C05479=1163.449,223.532,-63.405,-177.710,7.285,148.703
C05480=1163.454,223.284,-63.379,-177.713,7.282,148.703
C05481=1163.458,223.036,-63.354,-177.715,7.280,148.703
C05482=1163.463,222.787,-63.329,-177.718,7.278,148.704
C05483=1163.468,222.538,-63.303,-177.721,7.275,148.704
C05484=1163.472,222.289,-63.277,-177.724,7.273,148.704
C05485=1163.477,222.041,-63.252,-177.726,7.271,148.704
C05486=1163.481,221.792,-63.227,-177.729,7.268,148.704
C05487=1163.486,221.544,-63.202,-177.732,7.265,148.705
C05488=1163.489,221.295,-63.177,-177.734,7.263,148.705
C05489=1163.494,221.046,-63.151,-177.738,7.260,148.705
C05490=1163.499,220.798,-63.126,-177.740,7.258,148.705
C05491=1163.503,220.549,-63.100,-177.743,7.256,148.706
C05492=1163.508,220.300,-63.076,-177.745,7.254,148.706
C05493=1163.512,220.051,-63.050,-177.748,7.251,148.706
C05494=1163.517,219.803,-63.025,-177.751,7.248,148.706
C05495=1163.522,219.554,-63.000,-177.753,7.246,148.706
C05496=1163.525,219.305,-62.974,-177.757,7.243,148.706
C05497=1163.530,219.057,-62.949,-177.759,7.241,148.707
C05498=1163.535,218.808,-62.924,-177.762,7.239,148.707
C05499=1163.539,218.560,-62.899,-177.764,7.237,148.707
C05500=1163.544,218.310,-62.874,-177.767,7.234,148.707
C05501=1163.548,218.062,-62.849,-177.770,7.232,148.707
C05502=1163.553,217.813,-62.824,-177.772,7.229,148.708
C05503=1163.557,217.565,-62.798,-177.775,7.227,148.708
C05504=1163.562,217.315,-62.773,-177.778,7.224,148.708
C05505=1163.567,217.067,-62.748,-177.781,7.222,148.708
C05506=1163.571,216.818,-62.723,-177.783,7.219,148.708
C05507=1163.575,216.570,-62.698,-177.787,7.217,148.709
C05508=1163.580,216.321,-62.673,-177.789,7.215,148.709
C05509=1163.585,216.073,-62.648,-177.792,7.212,148.709
C05510=1163.589,215.823,-62.623,-177.794,7.210,148.709
C05511=1163.593,215.575,-62.598,-177.797,7.207,148.710
C05512=1163.598,215.326,-62.573,-177.800,7.205,148.710
C05513=1163.602,215.077,-62.549,-177.803,7.203,148.710
C05514=1163.607,214.829,-62.523,-177.805,7.201,148.710
C05515=1163.612,214.580,-62.498,-177.808,7.198,148.710
C05516=1163.616,214.331,-62.473,-177.811,7.196,148.711
C05517=1163.620,214.083,-62.448,-177.814,7.193,148.711
C05518=1163.625,213.834,-62.424,-177.816,7.191,148.711
C05519=1163.630,213.585,-62.398,-177.819,7.189,148.711
C05520=1163.634,213.337,-62.374,-177.821,7.186,148.711
C05521=1163.639,213.087,-62.349,-177.825,7.184,148.712
C05522=1163.644,212.839,-62.324,-177.827,7.182,148.712
C05523=1163.647,212.590,-62.299,-177.830,7.179,148.712
C05524=1163.652,212.341,-62.274,-177.832,7.177,148.712
C05525=1163.657,212.093,-62.250,-177.836,7.174,148.713
C05526=1163.661,211.844,-62.225,-177.838,7.172,148.713
C05527=1163.666,211.595,-62.200,-177.841,7.170,148.713
C05528=1163.670,211.346,-62.175,-177.843,7.168,148.713
C05529=1163.675,211.098,-62.151,-177.846,7.165,148.713
C05530=1163.679,210.849,-62.127,-177.849,7.163,148.714
C05531=1163.684,210.600,-62.101,-177.852,7.160,148.714
C05532=1163.689,210.330,-62.075,-177.854,7.158,148.714
C05533=1163.694,210.059,-62.048,-177.857,7.156,148.714
C05534=1163.699,209.789,-62.021,-177.861,7.153,148.715
C05535=1163.704,209.518,-61.994,-177.863,7.150,148.715
C05536=1163.708,209.269,-61.970,-177.866,7.148,148.715
C05537=1163.713,209.021,-61.945,-177.869,7.145,148.715
C05538=1163.717,208.772,-61.921,-177.872,7.144,148.716
C05539=1163.722,208.523,-61.896,-177.874,7.141,148.716
C05540=1163.726,208.275,-61.871,-177.877,7.139,148.716
C05541=1163.731,208.026,-61.847,-177.879,7.137,148.716
C05542=1163.735,207.777,-61.822,-177.882,7.134,148.716
C05543=1163.740,207.528,-61.798,-177.885,7.132,148.717
C05544=1163.744,207.280,-61.774,-177.888,7.129,148.717
C05545=1163.749,207.031,-61.749,-177.891,7.128,148.717
C05546=1163.753,206.782,-61.725,-177.893,7.125,148.717
C05547=1163.758,206.533,-61.700,-177.896,7.123,148.718
C05548=1163.763,206.285,-61.676,-177.899,7.120,148.718
C05549=1163.767,206.036,-61.651,-177.901,7.118,148.718
C05550=1163.772,205.787,-61.627,-177.904,7.115,148.718
C05551=1163.776,205.538,-61.603,-177.907,7.113,148.719
C05552=1163.782,205.289,-61.579,-177.909,7.111,148.719
C05553=1163.785,205.040,-61.554,-177.912,7.109,148.719
C05554=1163.790,204.792,-61.530,-177.915,7.107,148.719
C05555=1163.795,204.543,-61.505,-177.918,7.104,148.719
C05556=1163.799,204.295,-61.481,-177.920,7.102,148.720
C05557=1163.804,204.045,-61.456,-177.923,7.099,148.720
C05558=1163.808,203.797,-61.432,-177.926,7.098,148.720
C05559=1163.813,203.548,-61.409,-177.928,7.095,148.720
C05560=1163.817,203.299,-61.385,-177.931,7.093,148.721
C05561=1163.822,203.050,-61.360,-177.934,7.091,148.721
C05562=1163.826,202.802,-61.336,-177.937,7.088,148.721
C05563=1163.831,202.553,-61.312,-177.939,7.086,148.721
C05564=1163.836,202.304,-61.288,-177.942,7.083,148.722
C05565=1163.840,202.055,-61.264,-177.945,7.082,148.722
C05566=1163.844,201.806,-61.239,-177.948,7.080,148.722
C05567=1163.849,201.558,-61.215,-177.950,7.077,148.722
C05568=1163.854,201.309,-61.191,-177.953,7.075,148.723
C05569=1163.858,201.060,-61.167,-177.956,7.072,148.723
C05570=1163.863,200.812,-61.143,-177.959,7.071,148.723
C05571=1163.868,200.563,-61.120,-177.961,7.069,148.724
C05572=1163.872,200.313,-61.095,-177.964,7.066,148.724
C05573=1163.876,200.065,-61.071,-177.967,7.064,148.724
C05574=1163.881,199.816,-61.047,-177.969,7.061,148.724
C05575=1163.886,199.567,-61.023,-177.972,7.059,148.724
C05576=1163.890,199.319,-60.999,-177.975,7.058,148.725
C05577=1163.895,199.070,-60.975,-177.978,7.055,148.725
C05578=1163.899,198.821,-60.951,-177.980,7.053,148.725
C05579=1163.904,198.572,-60.927,-177.984,7.050,148.726
C05580=1163.908,198.323,-60.903,-177.986,7.048,148.726
C05581=1163.913,198.075,-60.879,-177.988,7.046,148.726
C05582=1163.917,197.826,-60.856,-177.991,7.043,148.726
C05583=1163.922,197.577,-60.831,-177.994,7.042,148.726
C05584=1163.927,197.328,-60.808,-177.997,7.039,148.727
C05585=1163.932,197.080,-60.784,-177.999,7.037,148.727
C05586=1163.936,196.831,-60.760,-178.002,7.035,148.727
C05587=1163.941,196.582,-60.736,-178.005,7.033,148.728
C05588=1163.945,196.332,-60.713,-178.007,7.031,148.728
C05589=1163.949,196.084,-60.688,-178.010,7.029,148.728
C05590=1163.954,195.835,-60.665,-178.013,7.026,148.728
C05591=1163.958,195.587,-60.641,-178.016,7.024,148.729
C05592=1163.964,195.337,-60.617,-178.019,7.022,148.729
C05593=1163.968,195.088,-60.594,-178.021,7.019,148.729
C05594=1163.973,194.840,-60.570,-178.024,7.018,148.729
C05595=1163.977,194.591,-60.546,-178.027,7.015,148.730
C05596=1163.982,194.342,-60.522,-178.029,7.013,148.730
C05597=1163.987,194.093,-60.499,-178.032,7.011,148.730
C05598=1163.991,193.844,-60.475,-178.035,7.009,148.730
C05599=1163.996,193.596,-60.451,-178.037,7.006,148.731
C05600=1164.000,193.347,-60.428,-178.040,7.005,148.731
C05601=1164.005,193.098,-60.405,-178.043,7.002,148.731
C05602=1164.009,192.849,-60.381,-178.045,7.000,148.731
C05603=1164.014,192.600,-60.357,-178.049,6.997,148.732
C05604=1164.019,192.351,-60.334,-178.051,6.996,148.732
C05605=1164.024,192.102,-60.311,-178.054,6.994,148.732
C05606=1164.028,191.854,-60.286,-178.057,6.991,148.733
C05607=1164.033,191.605,-60.263,-178.060,6.989,148.733
C05608=1164.037,191.356,-60.240,-178.062,6.987,148.733
C05609=1164.042,191.107,-60.216,-178.065,6.985,148.733
C05610=1164.046,190.859,-60.193,-178.068,6.983,148.734
C05611=1164.050,190.610,-60.170,-178.070,6.981,148.734
C05612=1164.055,190.361,-60.146,-178.073,6.978,148.734
C05613=1164.060,190.112,-60.123,-178.076,6.976,148.735
C05614=1164.065,189.862,-60.099,-178.078,6.975,148.735
C05615=1164.069,189.614,-60.075,-178.081,6.972,148.735
C05616=1164.074,189.365,-60.052,-178.084,6.970,148.735
C05617=1164.078,189.116,-60.029,-178.087,6.968,148.736
C05618=1164.083,188.867,-60.005,-178.089,6.965,148.736
C05619=1164.087,188.618,-59.983,-178.092,6.963,148.736
C05620=1164.092,188.370,-59.960,-178.095,6.962,148.737
C05621=1164.097,188.121,-59.936,-178.098,6.959,148.737
C05622=1164.102,187.872,-59.913,-178.100,6.957,148.737
C05623=1164.106,187.623,-59.889,-178.103,6.955,148.737
C05624=1164.111,187.374,-59.866,-178.106,6.953,148.738
C05625=1164.115,187.125,-59.843,-178.108,6.950,148.738
C05626=1164.120,186.876,-59.820,-178.111,6.949,148.738
C05627=1164.124,186.627,-59.797,-178.114,6.947,148.739
C05628=1164.129,186.378,-59.773,-178.117,6.944,148.739
C05629=1164.134,186.129,-59.750,-178.119,6.942,148.739
C05630=1164.138,185.881,-59.728,-178.122,6.940,148.739
C05631=1164.143,185.632,-59.704,-178.125,6.938,148.740
C05632=1164.148,185.383,-59.681,-178.127,6.936,148.740
C05633=1164.153,185.134,-59.657,-178.130,6.934,148.740
C05634=1164.156,184.885,-59.635,-178.133,6.932,148.741
C05635=1164.161,184.636,-59.611,-178.136,6.930,148.741
C05636=1164.166,184.366,-59.586,-178.138,6.928,148.741
C05637=1164.171,184.097,-59.562,-178.141,6.925,148.741
C05638=1164.176,183.828,-59.536,-178.144,6.923,148.742
C05639=1164.181,183.558,-59.511,-178.147,6.921,148.742
C05640=1164.185,183.309,-59.488,-178.150,6.919,148.742
C05641=1164.190,183.060,-59.466,-178.153,6.916,148.743
C05642=1164.196,182.811,-59.443,-178.156,6.914,148.743
C05643=1164.200,182.563,-59.420,-178.158,6.912,148.743
C05644=1164.204,182.313,-59.397,-178.161,6.911,148.744
C05645=1164.209,182.064,-59.373,-178.164,6.908,148.744
C05646=1164.213,181.816,-59.350,-178.166,6.906,148.744
C05647=1164.219,181.567,-59.328,-178.169,6.904,148.745
C05648=1164.223,181.318,-59.305,-178.172,6.903,148.745
C05649=1164.227,181.069,-59.282,-178.175,6.900,148.745
C05650=1164.232,180.820,-59.259,-178.177,6.898,148.745
C05651=1164.237,180.571,-59.237,-178.180,6.896,148.746
C05652=1164.242,180.322,-59.214,-178.183,6.894,148.746
C05653=1164.245,180.074,-59.191,-178.186,6.892,148.746
C05654=1164.250,179.824,-59.168,-178.189,6.890,148.747
C05655=1164.256,179.576,-59.145,-178.191,6.888,148.747
C05656=1164.260,179.327,-59.122,-178.194,6.885,148.747
C05657=1164.265,179.077,-59.100,-178.197,6.884,148.748
C05658=1164.269,178.829,-59.077,-178.199,6.882,148.748
C05659=1164.274,178.580,-59.054,-178.202,6.880,148.748
C05660=1164.278,178.331,-59.032,-178.205,6.877,148.748
C05661=1164.283,178.082,-59.009,-178.208,6.875,148.749
C05662=1164.287,177.833,-58.986,-178.210,6.874,148.749
C05663=1164.293,177.584,-58.964,-178.213,6.872,148.750
C05664=1164.297,177.335,-58.941,-178.215,6.870,148.750
C05665=1164.302,177.086,-58.918,-178.218,6.867,148.750
C05666=1164.306,176.838,-58.896,-178.221,6.865,148.750
C05667=1164.311,176.588,-58.873,-178.224,6.864,148.751
C05668=1164.315,176.339,-58.850,-178.226,6.862,148.751
C05669=1164.321,176.090,-58.828,-178.229,6.859,148.751
C05670=1164.325,175.842,-58.805,-178.232,6.857,148.752
C05671=1164.330,175.592,-58.783,-178.235,6.855,148.752
C05672=1164.334,175.344,-58.760,-178.237,6.854,148.752
C05673=1164.338,175.095,-58.738,-178.241,6.851,148.753
C05674=1164.343,174.846,-58.715,-178.243,6.849,148.753
C05675=1164.348,174.597,-58.693,-178.245,6.847,148.753
C05676=1164.353,174.348,-58.670,-178.248,6.845,148.754
C05677=1164.357,174.099,-58.648,-178.251,6.844,148.754
C05678=1164.362,173.850,-58.626,-178.254,6.841,148.754
C05679=1164.367,173.601,-58.603,-178.257,6.839,148.755
C05680=1164.371,173.352,-58.581,-178.259,6.837,148.755
C05681=1164.376,173.103,-58.558,-178.262,6.836,148.755
C05682=1164.380,172.854,-58.536,-178.264,6.834,148.756
C05683=1164.385,172.605,-58.514,-178.268,6.831,148.756
C05684=1164.390,172.356,-58.491,-178.270,6.829,148.756
C05685=1164.394,172.107,-58.469,-178.273,6.828,148.757
C05686=1164.399,171.858,-58.447,-178.275,6.826,148.757
C05687=1164.404,171.609,-58.424,-178.278,6.824,148.757
C05688=1164.409,171.361,-58.402,-178.281,6.821,148.757
C05689=1164.413,171.111,-58.380,-178.284,6.820,148.758
C05690=1164.418,170.863,-58.357,-178.287,6.818,148.758
C05691=1164.423,170.614,-58.335,-178.289,6.816,148.759
C05692=1164.427,170.364,-58.313,-178.292,6.814,148.759
C05693=1164.432,170.116,-58.291,-178.295,6.811,148.759
C05694=1164.437,169.866,-58.268,-178.297,6.810,148.759
C05695=1164.441,169.618,-58.246,-178.300,6.808,148.760
C05696=1164.445,169.369,-58.224,-178.303,6.806,148.760
C05697=1164.450,169.120,-58.202,-178.306,6.804,148.761
C05698=1164.455,168.870,-58.180,-178.308,6.803,148.761
C05699=1164.460,168.622,-58.158,-178.311,6.800,148.761
C05700=1164.464,168.373,-58.135,-178.314,6.798,148.761
C05701=1164.469,168.124,-58.114,-178.316,6.796,148.762
C05702=1164.473,167.875,-58.091,-178.319,6.794,148.762
C05703=1164.479,167.626,-58.069,-178.322,6.793,148.762
C05704=1164.483,167.377,-58.047,-178.324,6.791,148.763
C05705=1164.488,167.128,-58.025,-178.328,6.788,148.763
C05706=1164.492,166.879,-58.003,-178.330,6.787,148.764
C05707=1164.497,166.630,-57.982,-178.333,6.785,148.764
C05708=1164.502,166.380,-57.959,-178.335,6.783,148.764
C05709=1164.507,166.132,-57.937,-178.338,6.781,148.764
C05710=1164.511,165.883,-57.915,-178.341,6.779,148.765
C05711=1164.516,165.634,-57.893,-178.344,6.777,148.765
C05712=1164.520,165.385,-57.871,-178.347,6.775,148.766
C05713=1164.525,165.136,-57.849,-178.349,6.773,148.766
C05714=1164.529,164.887,-57.827,-178.352,6.771,148.766
C05715=1164.534,164.638,-57.805,-178.355,6.770,148.767
C05716=1164.538,164.389,-57.783,-178.357,6.768,148.767
C05717=1164.544,164.140,-57.761,-178.360,6.766,148.767
C05718=1164.549,163.890,-57.740,-178.363,6.763,148.768
C05719=1164.554,163.642,-57.718,-178.366,6.762,148.768
C05720=1164.558,163.393,-57.696,-178.368,6.760,148.768
C05721=1164.563,163.144,-57.674,-178.371,6.758,148.769
C05722=1164.568,162.895,-57.653,-178.374,6.756,148.769
C05723=1164.572,162.646,-57.631,-178.376,6.755,148.769
C05724=1164.577,162.397,-57.609,-178.379,6.753,148.770
C05725=1164.582,162.148,-57.587,-178.382,6.751,148.770
C05726=1164.586,161.899,-57.565,-178.385,6.748,148.771
C05727=1164.591,161.650,-57.544,-178.387,6.746,148.771
C05728=1164.595,161.400,-57.522,-178.390,6.745,148.771
C05729=1164.600,161.152,-57.501,-178.393,6.743,148.771
C05730=1164.605,160.903,-57.479,-178.395,6.741,148.772
C05731=1164.609,160.654,-57.457,-178.398,6.739,148.772
C05732=1164.614,160.405,-57.435,-178.401,6.738,148.773
C05733=1164.619,160.155,-57.414,-178.403,6.736,148.773
C05734=1164.624,159.907,-57.392,-178.407,6.733,148.773
C05735=1164.628,159.658,-57.370,-178.409,6.732,148.774
C05736=1164.633,159.409,-57.348,-178.412,6.730,148.774
C05737=1164.638,159.159,-57.327,-178.415,6.728,148.774
C05738=1164.642,158.911,-57.306,-178.417,6.726,148.775
C05739=1164.646,158.662,-57.284,-178.420,6.725,148.775
C05740=1164.652,158.392,-57.261,-178.423,6.723,148.776
C05741=1164.657,158.124,-57.239,-178.426,6.720,148.776
C05742=1164.662,157.855,-57.214,-178.429,6.719,148.776
C05743=1164.667,157.586,-57.192,-178.432,6.717,148.777
C05744=1164.671,157.337,-57.170,-178.435,6.714,148.777
C05745=1164.676,157.088,-57.149,-178.437,6.712,148.777
C05746=1164.681,156.839,-57.127,-178.440,6.711,148.778
C05747=1164.686,156.590,-57.105,-178.443,6.709,148.778
C05748=1164.691,156.340,-57.084,-178.446,6.707,148.778
C05749=1164.695,156.092,-57.063,-178.448,6.706,148.779
C05750=1164.700,155.843,-57.042,-178.451,6.704,148.779
C05751=1164.704,155.593,-57.020,-178.454,6.702,148.780
C05752=1164.710,155.344,-56.999,-178.456,6.700,148.780
C05753=1164.714,155.095,-56.977,-178.459,6.698,148.780
C05754=1164.719,154.847,-56.956,-178.461,6.696,148.781
C05755=1164.723,154.597,-56.935,-178.464,6.695,148.781
C05756=1164.728,154.349,-56.913,-178.467,6.693,148.781
C05757=1164.733,154.099,-56.892,-178.470,6.690,148.782
C05758=1164.738,153.851,-56.870,-178.473,6.689,148.782
C05759=1164.742,153.601,-56.850,-178.475,6.687,148.782
C05760=1164.747,153.352,-56.828,-178.478,6.685,148.783
C05761=1164.752,153.103,-56.807,-178.481,6.683,148.783
C05762=1164.757,152.854,-56.786,-178.483,6.682,148.784
C05763=1164.761,152.605,-56.765,-178.486,6.680,148.784
C05764=1164.766,152.356,-56.744,-178.489,6.678,148.784
C05765=1164.771,152.107,-56.722,-178.492,6.676,148.785
C05766=1164.776,151.858,-56.701,-178.494,6.675,148.785
C05767=1164.780,151.609,-56.680,-178.497,6.673,148.785
C05768=1164.785,151.360,-56.659,-178.500,6.671,148.786
C05769=1164.790,151.110,-56.638,-178.502,6.669,148.786
C05770=1164.794,150.862,-56.617,-178.505,6.668,148.787
C05771=1164.799,150.612,-56.596,-178.508,6.666,148.787
C05772=1164.804,150.363,-56.575,-178.510,6.664,148.787
C05773=1164.808,150.115,-56.554,-178.513,6.663,148.788
C05774=1164.813,149.866,-56.533,-178.516,6.661,148.788
C05775=1164.818,149.616,-56.511,-178.518,6.659,148.788
C05776=1164.822,149.367,-56.490,-178.522,6.656,148.789
C05777=1164.827,149.118,-56.469,-178.524,6.655,148.789
C05778=1164.833,148.869,-56.448,-178.527,6.653,148.790
C05779=1164.837,148.620,-56.428,-178.530,6.651,148.790
C05780=1164.842,148.371,-56.406,-178.533,6.650,148.790
C05781=1164.846,148.122,-56.386,-178.535,6.648,148.791
C05782=1164.851,147.872,-56.364,-178.538,6.646,148.791
C05783=1164.856,147.623,-56.344,-178.541,6.644,148.792
C05784=1164.860,147.374,-56.323,-178.543,6.643,148.792
C05785=1164.865,147.125,-56.301,-178.546,6.641,148.792
C05786=1164.870,146.877,-56.281,-178.549,6.639,148.793
C05787=1164.875,146.627,-56.260,-178.551,6.637,148.793
C05788=1164.879,146.378,-56.240,-178.554,6.636,148.793
C05789=1164.885,146.129,-56.219,-178.557,6.634,148.794
C05790=1164.889,145.880,-56.198,-178.560,6.632,148.794
C05791=1164.893,145.631,-56.176,-178.562,6.630,148.795
C05792=1164.898,145.382,-56.156,-178.565,6.629,148.795
C05793=1164.903,145.133,-56.135,-178.568,6.627,148.795
C05794=1164.907,144.884,-56.115,-178.570,6.625,148.796
C05795=1164.912,144.634,-56.094,-178.573,6.623,148.796
C05796=1164.917,144.385,-56.073,-178.576,6.622,148.797
C05797=1164.922,144.136,-56.052,-178.579,6.620,148.797
C05798=1164.927,143.887,-56.032,-178.582,6.619,148.797
C05799=1164.932,143.638,-56.011,-178.584,6.617,148.798
C05800=1164.936,143.389,-55.991,-178.587,6.615,148.798
C05801=1164.941,143.140,-55.970,-178.590,6.613,148.799
C05802=1164.946,142.891,-55.949,-178.592,6.612,148.799
C05803=1164.950,142.642,-55.929,-178.595,6.610,148.799
C05804=1164.955,142.393,-55.908,-178.598,6.608,148.800
C05805=1164.960,142.144,-55.888,-178.601,6.606,148.800
C05806=1164.965,141.894,-55.867,-178.603,6.605,148.801
C05807=1164.969,141.645,-55.846,-178.606,6.603,148.801
C05808=1164.974,141.396,-55.826,-178.609,6.601,148.801
C05809=1164.979,141.147,-55.805,-178.611,6.600,148.802
C05810=1164.983,140.898,-55.785,-178.614,6.598,148.802
C05811=1164.989,140.649,-55.764,-178.617,6.596,148.803
C05812=1164.993,140.400,-55.743,-178.619,6.594,148.803
C05813=1164.998,140.151,-55.723,-178.622,6.593,148.803
C05814=1165.003,139.901,-55.703,-178.625,6.592,148.804
C05815=1165.007,139.652,-55.682,-178.627,6.590,148.804
C05816=1165.012,139.403,-55.662,-178.630,6.589,148.805
C05817=1165.017,139.154,-55.641,-178.633,6.587,148.805
C05818=1165.021,138.905,-55.621,-178.636,6.585,148.805
C05819=1165.026,138.656,-55.600,-178.638,6.583,148.806
C05820=1165.031,138.406,-55.580,-178.641,6.582,148.806
C05821=1165.036,138.157,-55.560,-178.644,6.580,148.807
C05822=1165.040,137.908,-55.539,-178.646,6.578,148.807
C05823=1165.045,137.659,-55.519,-178.649,6.576,148.807
C05824=1165.050,137.410,-55.498,-178.652,6.575,148.808
C05825=1165.055,137.161,-55.478,-178.655,6.573,148.808
C05826=1165.060,136.912,-55.458,-178.657,6.571,148.809
C05827=1165.064,136.663,-55.438,-178.660,6.570,148.809
C05828=1165.069,136.414,-55.417,-178.663,6.568,148.810
C05829=1165.074,136.165,-55.397,-178.666,6.566,148.810
C05830=1165.078,135.916,-55.377,-178.669,6.565,148.810
C05831=1165.083,135.667,-55.356,-178.671,6.563,148.811
C05832=1165.088,135.417,-55.336,-178.674,6.561,148.811
C05833=1165.093,135.168,-55.316,-178.676,6.560,148.812
C05834=1165.097,134.919,-55.295,-178.679,6.559,148.812
C05835=1165.103,134.670,-55.276,-178.681,6.557,148.812
C05836=1165.107,134.421,-55.256,-178.684,6.555,148.813
C05837=1165.112,134.172,-55.235,-178.687,6.554,148.813
C05838=1165.117,133.922,-55.215,-178.690,6.552,148.814
C05839=1165.121,133.673,-55.195,-178.693,6.550,148.814
C05840=1165.126,133.424,-55.175,-178.695,6.549,148.814
C05841=1165.131,133.175,-55.155,-178.698,6.547,148.815
C05842=1165.136,132.926,-55.135,-178.701,6.545,148.815
C05843=1165.141,132.677,-55.114,-178.704,6.543,148.816
C05844=1165.146,132.408,-55.093,-178.706,6.542,148.816
C05845=1165.151,132.140,-55.072,-178.709,6.540,148.817
C05846=1165.156,131.871,-55.050,-178.712,6.538,148.817
C05847=1165.161,131.602,-55.029,-178.715,6.537,148.817
C05848=1165.166,131.353,-55.008,-178.718,6.535,148.818
C05849=1165.171,131.104,-54.988,-178.721,6.534,148.818
C05850=1165.176,130.855,-54.968,-178.724,6.532,148.819
C05851=1165.181,130.606,-54.949,-178.726,6.530,148.819
C05852=1165.185,130.357,-54.928,-178.729,6.528,148.820
C05853=1165.190,130.107,-54.908,-178.732,6.527,148.820
C05854=1165.195,129.858,-54.888,-178.734,6.525,148.820
C05855=1165.199,129.609,-54.868,-178.736,6.524,148.821
C05856=1165.205,129.360,-54.849,-178.739,6.522,148.821
C05857=1165.209,129.111,-54.829,-178.742,6.521,148.822
C05858=1165.214,128.861,-54.809,-178.745,6.519,148.822
C05859=1165.218,128.612,-54.789,-178.748,6.518,148.823
C05860=1165.224,128.363,-54.769,-178.750,6.516,148.823
C05861=1165.228,128.114,-54.750,-178.753,6.514,148.823
C05862=1165.233,127.865,-54.729,-178.756,6.512,148.824
C05863=1165.237,127.615,-54.710,-178.758,6.511,148.824
C05864=1165.243,127.367,-54.691,-178.761,6.510,148.825
C05865=1165.247,127.118,-54.670,-178.764,6.508,148.825
C05866=1165.252,126.868,-54.650,-178.767,6.507,148.826
C05867=1165.257,126.619,-54.631,-178.769,6.505,148.826
C05868=1165.262,126.370,-54.611,-178.772,6.503,148.826
C05869=1165.267,126.121,-54.591,-178.775,6.501,148.827
C05870=1165.271,125.871,-54.572,-178.778,6.500,148.827
C05871=1165.277,125.622,-54.552,-178.780,6.499,148.828
C05872=1165.280,125.374,-54.532,-178.783,6.497,148.828
C05873=1165.285,125.124,-54.513,-178.786,6.496,148.829
C05874=1165.290,124.875,-54.493,-178.788,6.494,148.829
C05875=1165.295,124.626,-54.474,-178.791,6.492,148.829
C05876=1165.300,124.377,-54.453,-178.794,6.491,148.830
C05877=1165.305,124.128,-54.434,-178.797,6.489,148.830
C05878=1165.310,123.878,-54.415,-178.799,6.488,148.831
C05879=1165.314,123.629,-54.395,-178.802,6.487,148.831
C05880=1165.319,123.380,-54.376,-178.804,6.485,148.832
C05881=1165.324,123.130,-54.357,-178.807,6.483,148.832
C05882=1165.328,122.882,-54.336,-178.810,6.482,148.833
C05883=1165.334,122.633,-54.317,-178.813,6.480,148.833
C05884=1165.338,122.383,-54.297,-178.815,6.479,148.834
C05885=1165.343,122.134,-54.278,-178.818,6.477,148.834
C05886=1165.348,121.885,-54.259,-178.821,6.476,148.834
C05887=1165.352,121.635,-54.239,-178.823,6.474,148.835
C05888=1165.357,121.386,-54.220,-178.826,6.473,148.835
C05889=1165.362,121.137,-54.200,-178.829,6.471,148.836
C05890=1165.367,120.887,-54.181,-178.831,6.470,148.836
C05891=1165.372,120.639,-54.162,-178.834,6.468,148.837
C05892=1165.377,120.389,-54.142,-178.837,6.467,148.837
C05893=1165.381,120.140,-54.123,-178.840,6.465,148.838
C05894=1165.387,119.891,-54.103,-178.843,6.463,148.838
C05895=1165.391,119.642,-54.084,-178.845,6.462,148.838
C05896=1165.396,119.393,-54.065,-178.847,6.461,148.839
C05897=1165.401,119.143,-54.045,-178.850,6.459,148.839
C05898=1165.406,118.894,-54.026,-178.853,6.458,148.840
C05899=1165.410,118.645,-54.007,-178.856,6.456,148.840
C05900=1165.415,118.395,-53.987,-178.859,6.454,148.841
C05901=1165.420,118.147,-53.968,-178.861,6.453,148.841
C05902=1165.425,117.897,-53.948,-178.864,6.452,148.841
C05903=1165.430,117.648,-53.930,-178.867,6.450,148.842
C05904=1165.434,117.399,-53.910,-178.870,6.449,148.842
C05905=1165.440,117.150,-53.891,-178.872,6.447,148.843
C05906=1165.444,116.901,-53.872,-178.875,6.445,148.843
C05907=1165.449,116.651,-53.853,-178.877,6.444,148.844
C05908=1165.454,116.402,-53.833,-178.880,6.443,148.844
C05909=1165.459,116.153,-53.815,-178.883,6.441,148.845
C05910=1165.463,115.904,-53.795,-178.886,6.439,148.845
C05911=1165.469,115.655,-53.776,-178.888,6.438,148.845
C05912=1165.473,115.405,-53.757,-178.891,6.437,148.846
C05913=1165.478,115.156,-53.738,-178.894,6.435,148.847
C05914=1165.482,114.907,-53.719,-178.896,6.434,148.847
C05915=1165.488,114.658,-53.700,-178.899,6.432,148.847
C05916=1165.492,114.408,-53.680,-178.901,6.431,148.848
C05917=1165.497,114.160,-53.661,-178.905,6.430,148.848
C05918=1165.502,113.910,-53.642,-178.907,6.428,148.849
C05919=1165.507,113.661,-53.624,-178.910,6.426,148.849
C05920=1165.511,113.411,-53.604,-178.913,6.425,148.850
C05921=1165.517,113.162,-53.586,-178.915,6.424,148.850
C05922=1165.521,112.913,-53.566,-178.918,6.422,148.851
C05923=1165.526,112.664,-53.547,-178.921,6.421,148.851
C05924=1165.530,112.415,-53.528,-178.923,6.419,148.851
C05925=1165.536,112.165,-53.510,-178.926,6.418,148.852
C05926=1165.540,111.916,-53.490,-178.929,6.417,148.852
C05927=1165.545,111.667,-53.471,-178.931,6.415,148.853
C05928=1165.550,111.418,-53.453,-178.934,6.413,148.853
C05929=1165.555,111.168,-53.434,-178.936,6.412,148.854
C05930=1165.560,110.920,-53.415,-178.940,6.411,148.854
C05931=1165.565,110.669,-53.396,-178.942,6.409,148.855
C05932=1165.569,110.421,-53.377,-178.945,6.408,148.855
C05933=1165.574,110.171,-53.358,-178.948,6.406,148.856
C05934=1165.579,109.922,-53.340,-178.950,6.405,148.856
C05935=1165.585,109.673,-53.321,-178.953,6.404,148.857
C05936=1165.589,109.423,-53.302,-178.956,6.402,148.857
C05937=1165.594,109.175,-53.283,-178.958,6.400,148.857
C05938=1165.598,108.925,-53.264,-178.961,6.400,148.858
C05939=1165.603,108.676,-53.246,-178.964,6.398,148.858
C05940=1165.609,108.427,-53.227,-178.966,6.396,148.859
C05941=1165.613,108.177,-53.208,-178.969,6.395,148.859
C05942=1165.618,107.928,-53.189,-178.972,6.394,148.860
C05943=1165.623,107.679,-53.171,-178.975,6.392,148.860
C05944=1165.628,107.429,-53.152,-178.977,6.390,148.861
C05945=1165.632,107.181,-53.133,-178.979,6.390,148.861
C05946=1165.637,106.931,-53.115,-178.983,6.388,148.862
C05947=1165.642,106.682,-53.095,-178.985,6.387,148.862
C05948=1165.647,106.414,-53.076,-178.988,6.385,148.863
C05949=1165.653,106.145,-53.056,-178.991,6.383,148.863
C05950=1165.657,105.877,-53.036,-178.994,6.382,148.864
C05951=1165.663,105.608,-53.016,-178.997,6.380,148.864
C05952=1165.668,105.359,-52.998,-178.999,6.379,148.865
C05953=1165.673,105.110,-52.979,-179.002,6.378,148.865
C05954=1165.678,104.860,-52.960,-179.005,6.376,148.866
C05955=1165.683,104.611,-52.942,-179.008,6.375,148.866
C05956=1165.687,104.362,-52.923,-179.010,6.374,148.867
C05957=1165.692,104.112,-52.904,-179.013,6.372,148.867
C05958=1165.697,103.863,-52.886,-179.016,6.371,148.868
C05959=1165.702,103.615,-52.868,-179.018,6.370,148.868
C05960=1165.707,103.364,-52.849,-179.021,6.368,148.868
C05961=1165.712,103.115,-52.831,-179.024,6.367,148.869
C05962=1165.716,102.867,-52.812,-179.026,6.366,148.869
C05963=1165.721,102.617,-52.794,-179.029,6.364,148.870
C05964=1165.726,102.367,-52.775,-179.032,6.362,148.870
C05965=1165.731,102.119,-52.756,-179.035,6.361,148.871
C05966=1165.736,101.870,-52.738,-179.037,6.360,148.871
C05967=1165.741,101.620,-52.720,-179.040,6.359,148.872
C05968=1165.746,101.370,-52.702,-179.043,6.357,148.872
C05969=1165.750,101.122,-52.683,-179.045,6.356,148.873
C05970=1165.755,100.872,-52.665,-179.048,6.355,148.873
C05971=1165.760,100.623,-52.647,-179.051,6.353,148.874
C05972=1165.764,100.373,-52.629,-179.053,6.352,148.874
C05973=1165.770,100.124,-52.610,-179.056,6.351,148.875
C05974=1165.775,99.875,-52.592,-179.058,6.349,148.875
C05975=1165.780,99.626,-52.573,-179.061,6.348,148.876
C05976=1165.784,99.376,-52.555,-179.064,6.347,148.876
C05977=1165.789,99.127,-52.537,-179.067,6.345,148.877
C05978=1165.794,98.878,-52.518,-179.069,6.344,148.877
C05979=1165.799,98.628,-52.500,-179.072,6.343,148.878
C05980=1165.804,98.379,-52.482,-179.075,6.341,148.878
C05981=1165.809,98.129,-52.464,-179.078,6.340,148.879
C05982=1165.814,97.880,-52.446,-179.080,6.339,148.879
C05983=1165.818,97.632,-52.427,-179.083,6.337,148.880
C05984=1165.823,97.382,-52.409,-179.086,6.336,148.880
C05985=1165.828,97.133,-52.391,-179.088,6.335,148.881
C05986=1165.834,96.884,-52.373,-179.091,6.333,148.881
C05987=1165.838,96.634,-52.354,-179.093,6.331,148.881
C05988=1165.843,96.385,-52.337,-179.096,6.331,148.882
C05989=1165.848,96.136,-52.319,-179.099,6.329,148.882
C05990=1165.853,95.886,-52.301,-179.101,6.328,148.883
C05991=1165.858,95.637,-52.283,-179.104,6.327,148.884
C05992=1165.862,95.388,-52.265,-179.107,6.325,148.884
C05993=1165.867,95.139,-52.247,-179.109,6.324,148.884
C05994=1165.872,94.889,-52.228,-179.112,6.323,148.885
C05995=1165.877,94.640,-52.210,-179.115,6.321,148.885
C05996=1165.882,94.391,-52.192,-179.117,6.320,148.886
C05997=1165.886,94.141,-52.174,-179.120,6.319,148.887
C05998=1165.891,93.892,-52.156,-179.123,6.317,148.887
C05999=1165.897,93.643,-52.139,-179.125,6.316,148.887
C06000=1165.901,93.393,-52.121,-179.128,6.315,148.888
C06001=1165.906,93.144,-52.103,-179.131,6.313,148.888
C06002=1165.911,92.895,-52.085,-179.133,6.313,148.889
C06003=1165.916,92.645,-52.067,-179.136,6.311,148.889
C06004=1165.921,92.396,-52.049,-179.139,6.310,148.890
C06005=1165.925,92.147,-52.031,-179.141,6.309,148.890
C06006=1165.930,91.898,-52.013,-179.145,6.307,148.891
C06007=1165.936,91.648,-51.996,-179.147,6.306,148.891
C06008=1165.940,91.399,-51.978,-179.149,6.305,148.892
C06009=1165.945,91.149,-51.960,-179.153,6.303,148.892
C06010=1165.950,90.900,-51.942,-179.155,6.302,148.893
C06011=1165.955,90.651,-51.924,-179.158,6.301,148.893
C06012=1165.960,90.401,-51.906,-179.160,6.300,148.894
C06013=1165.965,90.152,-51.888,-179.163,6.299,148.894
C06014=1165.970,89.903,-51.871,-179.166,6.297,148.895
C06015=1165.974,89.654,-51.853,-179.168,6.296,148.895
C06016=1165.979,89.405,-51.835,-179.171,6.295,148.896
C06017=1165.985,89.155,-51.818,-179.174,6.293,148.896
C06018=1165.989,88.906,-51.800,-179.176,6.292,148.897
C06019=1165.994,88.657,-51.782,-179.179,6.291,148.897
C06020=1166.000,88.407,-51.765,-179.182,6.290,148.898
C06021=1166.005,88.158,-51.747,-179.184,6.288,148.898
C06022=1166.009,87.909,-51.729,-179.187,6.287,148.899
C06023=1166.014,87.659,-51.712,-179.190,6.286,148.899
C06024=1166.019,87.410,-51.694,-179.192,6.285,148.900
C06025=1166.024,87.161,-51.676,-179.195,6.284,148.901
C06026=1166.029,86.911,-51.659,-179.198,6.282,148.901
C06027=1166.034,86.662,-51.641,-179.200,6.281,148.901
C06028=1166.038,86.413,-51.623,-179.203,6.280,148.902
C06029=1166.043,86.163,-51.606,-179.206,6.278,148.902
C06030=1166.048,85.914,-51.588,-179.208,6.278,148.903
C06031=1166.053,85.665,-51.570,-179.211,6.276,148.904
C06032=1166.058,85.415,-51.553,-179.213,6.275,148.904
C06033=1166.062,85.166,-51.536,-179.216,6.274,148.904
C06034=1166.068,84.916,-51.518,-179.219,6.272,148.905
C06035=1166.073,84.667,-51.500,-179.221,6.271,148.905
C06036=1166.078,84.417,-51.483,-179.225,6.270,148.906
C06037=1166.082,84.169,-51.466,-179.227,6.269,148.907
C06038=1166.087,83.919,-51.448,-179.229,6.267,148.907
C06039=1166.092,83.670,-51.430,-179.233,6.266,148.908
C06040=1166.097,83.420,-51.413,-179.235,6.265,148.908
C06041=1166.102,83.171,-51.396,-179.238,6.264,148.909
C06042=1166.107,82.921,-51.378,-179.240,6.263,148.909
C06043=1166.112,82.672,-51.360,-179.243,6.261,148.910
C06044=1166.117,82.423,-51.344,-179.246,6.261,148.910
C06045=1166.122,82.174,-51.326,-179.248,6.259,148.911
C06046=1166.127,81.924,-51.309,-179.250,6.258,148.911
C06047=1166.132,81.675,-51.291,-179.254,6.257,148.912
C06048=1166.136,81.425,-51.274,-179.256,6.255,148.912
C06049=1166.141,81.176,-51.256,-179.259,6.255,148.913
C06050=1166.146,80.927,-51.239,-179.262,6.253,148.913
C06051=1166.151,80.677,-51.222,-179.264,6.252,148.914
C06052=1166.157,80.409,-51.203,-179.267,6.251,148.914
C06053=1166.162,80.141,-51.185,-179.270,6.249,148.915
C06054=1166.167,79.872,-51.167,-179.272,6.249,148.915
C06055=1166.173,79.604,-51.148,-179.276,6.247,148.916
C06056=1166.177,79.355,-51.130,-179.278,6.246,148.916
C06057=1166.182,79.105,-51.114,-179.281,6.245,148.917
C06058=1166.187,78.855,-51.096,-179.284,6.243,148.917
C06059=1166.191,78.607,-51.079,-179.286,6.242,148.918
C06060=1166.197,78.357,-51.062,-179.289,6.241,148.919
C06061=1166.202,78.108,-51.045,-179.291,6.240,148.919
C06062=1166.207,77.859,-51.027,-179.294,6.239,148.920
C06063=1166.212,77.609,-51.010,-179.297,6.237,148.920
C06064=1166.216,77.360,-50.993,-179.299,6.236,148.920
C06065=1166.221,77.110,-50.976,-179.303,6.235,148.921
C06066=1166.226,76.861,-50.959,-179.305,6.234,148.922
C06067=1166.231,76.612,-50.942,-179.308,6.233,148.922
C06068=1166.237,76.362,-50.925,-179.310,6.232,148.923
C06069=1166.241,76.112,-50.908,-179.313,6.230,148.923
C06070=1166.246,75.863,-50.890,-179.315,6.230,148.924
C06071=1166.251,75.615,-50.874,-179.318,6.228,148.924
C06072=1166.256,75.365,-50.856,-179.321,6.228,148.925
C06073=1166.261,75.115,-50.840,-179.323,6.226,148.925
C06074=1166.266,74.865,-50.822,-179.326,6.225,148.926
C06075=1166.270,74.617,-50.805,-179.329,6.224,148.926
C06076=1166.276,74.368,-50.788,-179.331,6.223,148.927
C06077=1166.281,74.118,-50.772,-179.334,6.221,148.927
C06078=1166.286,73.868,-50.754,-179.336,6.221,148.928
C06079=1166.290,73.619,-50.738,-179.340,6.219,148.928
C06080=1166.295,73.370,-50.721,-179.342,6.218,148.929
C06081=1166.301,73.120,-50.704,-179.344,6.217,148.929
C06082=1166.305,72.871,-50.687,-179.347,6.216,148.930
C06083=1166.310,72.621,-50.670,-179.350,6.214,148.930
C06084=1166.315,72.373,-50.653,-179.352,6.214,148.931
C06085=1166.320,72.123,-50.636,-179.355,6.212,148.932
C06086=1166.325,71.873,-50.619,-179.358,6.212,148.932
C06087=1166.330,71.625,-50.603,-179.361,6.210,148.933
C06088=1166.335,71.375,-50.586,-179.363,6.209,148.933
C06089=1166.340,71.125,-50.569,-179.366,6.208,148.934
C06090=1166.345,70.876,-50.552,-179.368,6.207,148.934
C06091=1166.350,70.627,-50.535,-179.371,6.206,148.935
C06092=1166.354,70.377,-50.519,-179.373,6.205,148.935
C06093=1166.360,70.128,-50.501,-179.377,6.203,148.936
C06094=1166.365,69.879,-50.485,-179.379,6.203,148.936
C06095=1166.369,69.629,-50.468,-179.382,6.201,148.937
C06096=1166.374,69.379,-50.451,-179.384,6.200,148.937
C06097=1166.379,69.131,-50.435,-179.387,6.199,148.938
C06098=1166.384,68.881,-50.418,-179.390,6.198,148.939
C06099=1166.389,68.631,-50.401,-179.392,6.196,148.939
C06100=1166.394,68.382,-50.385,-179.395,6.196,148.940
C06101=1166.399,68.133,-50.369,-179.398,6.194,148.940
C06102=1166.404,67.883,-50.351,-179.400,6.194,148.941
C06103=1166.409,67.634,-50.335,-179.402,6.193,148.941
C06104=1166.414,67.384,-50.318,-179.405,6.191,148.942
C06105=1166.419,67.135,-50.301,-179.408,6.191,148.942
C06106=1166.424,66.886,-50.285,-179.411,6.189,148.943
C06107=1166.428,66.636,-50.268,-179.413,6.189,148.943
C06108=1166.433,66.386,-50.252,-179.416,6.187,148.944
C06109=1166.439,66.137,-50.235,-179.419,6.186,148.944
C06110=1166.444,65.888,-50.219,-179.421,6.185,148.945
C06111=1166.449,65.639,-50.202,-179.424,6.184,148.945
C06112=1166.453,65.389,-50.186,-179.427,6.182,148.946
C06113=1166.458,65.140,-50.168,-179.429,6.182,148.947
C06114=1166.464,64.890,-50.153,-179.431,6.181,148.947
C06115=1166.468,64.641,-50.136,-179.434,6.179,148.947
C06116=1166.473,64.392,-50.120,-179.437,6.179,148.948
C06117=1166.478,64.142,-50.103,-179.440,6.177,148.949
C06118=1166.483,63.892,-50.087,-179.442,6.177,148.949
C06119=1166.488,63.643,-50.070,-179.445,6.175,148.950
C06120=1166.493,63.394,-50.054,-179.448,6.175,148.950
C06121=1166.498,63.145,-50.037,-179.450,6.173,148.951
C06122=1166.503,62.895,-50.021,-179.453,6.172,148.951
C06123=1166.509,62.646,-50.005,-179.455,6.171,148.952
C06124=1166.513,62.396,-49.988,-179.458,6.170,148.952
C06125=1166.518,62.146,-49.972,-179.460,6.169,148.953
C06126=1166.523,61.897,-49.956,-179.464,6.168,148.954
C06127=1166.527,61.648,-49.939,-179.466,6.167,148.954
C06128=1166.533,61.399,-49.923,-179.469,6.166,148.955
C06129=1166.537,61.149,-49.907,-179.471,6.165,148.955
C06130=1166.542,60.900,-49.890,-179.473,6.164,148.956
C06131=1166.548,60.650,-49.874,-179.477,6.163,148.956
C06132=1166.553,60.401,-49.858,-179.479,6.162,148.957
C06133=1166.558,60.151,-49.842,-179.482,6.161,148.957
C06134=1166.563,59.902,-49.825,-179.484,6.160,148.958
C06135=1166.567,59.653,-49.809,-179.487,6.158,148.958
C06136=1166.573,59.403,-49.793,-179.489,6.157,148.959
C06137=1166.577,59.154,-49.776,-179.492,6.157,148.960
C06138=1166.583,58.904,-49.761,-179.495,6.155,148.960
C06139=1166.587,58.655,-49.744,-179.497,6.155,148.961
C06140=1166.592,58.406,-49.728,-179.500,6.153,148.961
C06141=1166.597,58.156,-49.712,-179.503,6.153,148.962
C06142=1166.602,57.907,-49.696,-179.505,6.152,148.962
C06143=1166.607,57.657,-49.680,-179.508,6.150,148.963
C06144=1166.613,57.408,-49.663,-179.510,6.150,148.963
C06145=1166.617,57.158,-49.647,-179.514,6.148,148.964
C06146=1166.623,56.909,-49.631,-179.516,6.147,148.964
C06147=1166.627,56.659,-49.614,-179.518,6.147,148.965
C06148=1166.633,56.410,-49.599,-179.521,6.145,148.965
C06149=1166.638,56.161,-49.583,-179.524,6.145,148.966
C06150=1166.642,55.911,-49.567,-179.526,6.143,148.967
C06151=1166.648,55.662,-49.550,-179.529,6.143,148.967
C06152=1166.652,55.412,-49.534,-179.531,6.142,148.968
C06153=1166.657,55.163,-49.518,-179.534,6.140,148.968
C06154=1166.662,54.913,-49.502,-179.537,6.140,148.969
C06155=1166.667,54.664,-49.487,-179.539,6.139,148.969
C06156=1166.672,54.396,-49.469,-179.542,6.137,148.970
C06157=1166.678,54.128,-49.452,-179.545,6.136,148.971
C06158=1166.683,53.858,-49.435,-179.548,6.136,148.971
C06159=1166.688,53.590,-49.418,-179.551,6.134,148.972
C06160=1166.694,53.341,-49.402,-179.553,6.133,148.972
C06161=1166.698,53.091,-49.386,-179.555,6.132,148.973
C06162=1166.703,52.842,-49.370,-179.559,6.131,148.973
C06163=1166.709,52.592,-49.355,-179.561,6.130,148.974
C06164=1166.713,52.343,-49.338,-179.564,6.129,148.975
C06165=1166.719,52.093,-49.322,-179.566,6.128,148.975
C06166=1166.723,51.843,-49.306,-179.569,6.128,148.976
C06167=1166.729,51.594,-49.291,-179.572,6.126,148.976
C06168=1166.734,51.345,-49.274,-179.574,6.125,148.977
C06169=1166.738,51.095,-49.259,-179.576,6.125,148.977
C06170=1166.743,50.846,-49.243,-179.580,6.123,148.978
C06171=1166.749,50.596,-49.228,-179.582,6.122,148.978
C06172=1166.753,50.347,-49.211,-179.584,6.122,148.979
C06173=1166.759,50.098,-49.196,-179.587,6.120,148.979
C06174=1166.763,49.847,-49.180,-179.590,6.120,148.980
C06175=1166.768,49.598,-49.165,-179.592,6.119,148.981
C06176=1166.773,49.350,-49.148,-179.595,6.118,148.981
C06177=1166.778,49.100,-49.132,-179.597,6.117,148.982
C06178=1166.783,48.850,-49.117,-179.601,6.115,148.982
C06179=1166.789,48.601,-49.101,-179.603,6.115,148.983
C06180=1166.793,48.352,-49.086,-179.605,6.114,148.983
C06181=1166.798,48.102,-49.070,-179.608,6.112,148.984
C06182=1166.803,47.853,-49.054,-179.611,6.112,148.985
C06183=1166.809,47.603,-49.038,-179.613,6.111,148.985
C06184=1166.813,47.353,-49.022,-179.616,6.110,148.986
C06185=1166.818,47.104,-49.007,-179.618,6.109,148.986
C06186=1166.823,46.855,-48.992,-179.621,6.108,148.987
C06187=1166.828,46.605,-48.976,-179.624,6.107,148.987
C06188=1166.834,46.355,-48.960,-179.626,6.106,148.988
C06189=1166.838,46.106,-48.945,-179.628,6.105,148.988
C06190=1166.844,45.857,-48.930,-179.632,6.104,148.989
C06191=1166.848,45.607,-48.914,-179.634,6.103,148.989
C06192=1166.853,45.358,-48.898,-179.636,6.103,148.990
C06193=1166.858,45.109,-48.882,-179.639,6.102,148.991
C06194=1166.864,44.859,-48.867,-179.642,6.101,148.991
C06195=1166.868,44.609,-48.851,-179.644,6.100,148.992
C06196=1166.873,44.360,-48.836,-179.647,6.099,148.992
C06197=1166.878,44.111,-48.820,-179.650,6.098,148.993
C06198=1166.884,43.861,-48.805,-179.652,6.097,148.993
C06199=1166.888,43.612,-48.789,-179.655,6.097,148.994
C06200=1166.893,43.362,-48.774,-179.657,6.095,148.995
C06201=1166.899,43.113,-48.758,-179.660,6.094,148.995
C06202=1166.903,42.864,-48.743,-179.662,6.094,148.996
C06203=1166.908,42.614,-48.727,-179.665,6.092,148.996
C06204=1166.914,42.364,-48.712,-179.668,6.091,148.997
C06205=1166.918,42.114,-48.697,-179.670,6.091,148.997
C06206=1166.924,41.865,-48.682,-179.673,6.089,148.998
C06207=1166.928,41.616,-48.667,-179.676,6.089,148.999
C06208=1166.933,41.366,-48.651,-179.678,6.088,148.999
C06209=1166.939,41.116,-48.635,-179.680,6.087,149.000
C06210=1166.943,40.867,-48.620,-179.683,6.086,149.000
C06211=1166.949,40.618,-48.605,-179.686,6.085,149.001
C06212=1166.953,40.369,-48.590,-179.688,6.085,149.002
C06213=1166.959,40.119,-48.574,-179.691,6.083,149.002
C06214=1166.964,39.869,-48.559,-179.694,6.083,149.003
C06215=1166.968,39.620,-48.544,-179.696,6.082,149.003
C06216=1166.974,39.370,-48.528,-179.699,6.081,149.004
C06217=1166.978,39.121,-48.513,-179.701,6.080,149.004
C06218=1166.984,38.872,-48.498,-179.704,6.079,149.005
C06219=1166.989,38.622,-48.483,-179.706,6.078,149.005
C06220=1166.994,38.372,-48.468,-179.709,6.077,149.006
C06221=1166.999,38.123,-48.452,-179.712,6.076,149.006
C06222=1167.004,37.873,-48.437,-179.714,6.076,149.007
C06223=1167.009,37.624,-48.421,-179.716,6.075,149.008
C06224=1167.014,37.374,-48.407,-179.720,6.074,149.008
C06225=1167.019,37.125,-48.391,-179.722,6.073,149.009
C06226=1167.024,36.876,-48.376,-179.724,6.072,149.009
C06227=1167.029,36.626,-48.361,-179.727,6.072,149.010
C06228=1167.034,36.377,-48.347,-179.730,6.070,149.010
C06229=1167.039,36.127,-48.331,-179.732,6.070,149.011
C06230=1167.044,35.878,-48.316,-179.735,6.069,149.012
C06231=1167.049,35.628,-48.301,-179.738,6.067,149.012
C06232=1167.054,35.378,-48.286,-179.740,6.067,149.013
C06233=1167.059,35.129,-48.271,-179.743,6.066,149.013
C06234=1167.064,34.879,-48.256,-179.745,6.065,149.014
C06235=1167.069,34.630,-48.241,-179.748,6.064,149.015
C06236=1167.074,34.381,-48.225,-179.750,6.063,149.015
C06237=1167.079,34.131,-48.211,-179.753,6.063,149.016
C06238=1167.085,33.882,-48.196,-179.755,6.062,149.016
C06239=1167.089,33.633,-48.181,-179.758,6.060,149.017
C06240=1167.095,33.383,-48.166,-179.761,6.060,149.017
C06241=1167.099,33.133,-48.150,-179.763,6.059,149.018
C06242=1167.104,32.884,-48.135,-179.766,6.059,149.019
C06243=1167.110,32.634,-48.120,-179.768,6.057,149.019
C06244=1167.114,32.385,-48.105,-179.771,6.056,149.020
C06245=1167.119,32.135,-48.091,-179.773,6.056,149.020
C06246=1167.125,31.885,-48.076,-179.776,6.055,149.021
C06247=1167.129,31.636,-48.061,-179.779,6.054,149.021
C06248=1167.135,31.386,-48.046,-179.781,6.053,149.022
C06249=1167.140,31.137,-48.031,-179.784,6.053,149.023
C06250=1167.144,30.888,-48.016,-179.786,6.052,149.023
C06251=1167.150,30.638,-48.001,-179.789,6.051,149.024
C06252=1167.155,30.388,-47.987,-179.791,6.050,149.024
C06253=1167.159,30.139,-47.972,-179.794,6.049,149.025
C06254=1167.165,29.889,-47.957,-179.796,6.048,149.025
C06255=1167.170,29.640,-47.942,-179.799,6.048,149.026
C06256=1167.175,29.391,-47.927,-179.802,6.046,149.027
C06257=1167.180,29.141,-47.913,-179.804,6.046,149.027
C06258=1167.185,28.891,-47.898,-179.807,6.045,149.028
C06259=1167.190,28.642,-47.883,-179.809,6.044,149.028
C06260=1167.196,28.373,-47.867,-179.812,6.043,149.029
C06261=1167.201,28.104,-47.851,-179.815,6.042,149.030
C06262=1167.206,27.835,-47.836,-179.818,6.042,149.030
C06263=1167.212,27.566,-47.819,-179.820,6.040,149.031
C06264=1167.217,27.317,-47.804,-179.823,6.040,149.031
C06265=1167.222,27.067,-47.790,-179.825,6.039,149.032
C06266=1167.227,26.818,-47.776,-179.828,6.039,149.033
C06267=1167.233,26.569,-47.760,-179.831,6.037,149.033
C06268=1167.238,26.319,-47.746,-179.833,6.036,149.034
C06269=1167.242,26.070,-47.731,-179.836,6.036,149.034
C06270=1167.247,25.820,-47.717,-179.838,6.035,149.035
C06271=1167.253,25.570,-47.702,-179.841,6.035,149.035
C06272=1167.257,25.321,-47.687,-179.843,6.033,149.036
C06273=1167.262,25.071,-47.673,-179.846,6.033,149.037
C06274=1167.267,24.822,-47.659,-179.848,6.032,149.037
C06275=1167.272,24.572,-47.644,-179.851,6.031,149.038
C06276=1167.278,24.323,-47.629,-179.854,6.031,149.038
C06277=1167.283,24.073,-47.614,-179.856,6.029,149.039
C06278=1167.288,23.823,-47.600,-179.859,6.029,149.040
C06279=1167.293,23.575,-47.585,-179.861,6.028,149.040
C06280=1167.298,23.325,-47.571,-179.864,6.027,149.041
C06281=1167.303,23.075,-47.557,-179.866,6.026,149.041
C06282=1167.308,22.826,-47.543,-179.869,6.025,149.042
C06283=1167.313,22.576,-47.527,-179.872,6.025,149.043
C06284=1167.318,22.326,-47.513,-179.874,6.024,149.043
C06285=1167.323,22.077,-47.499,-179.877,6.023,149.044
C06286=1167.328,21.827,-47.484,-179.879,6.022,149.044
C06287=1167.333,21.577,-47.470,-179.882,6.021,149.045
C06288=1167.338,21.329,-47.455,-179.884,6.020,149.045
C06289=1167.343,21.079,-47.441,-179.887,6.020,149.046
C06290=1167.348,20.830,-47.427,-179.890,6.019,149.047
C06291=1167.354,20.580,-47.412,-179.892,6.019,149.047
C06292=1167.359,20.330,-47.398,-179.894,6.018,149.048
C06293=1167.364,20.080,-47.383,-179.897,6.016,149.048
C06294=1167.369,19.832,-47.369,-179.900,6.016,149.049
C06295=1167.374,19.582,-47.354,-179.902,6.015,149.049
C06296=1167.379,19.332,-47.340,-179.905,6.015,149.050
C06297=1167.384,19.083,-47.326,-179.907,6.014,149.051
C06298=1167.389,18.833,-47.312,-179.909,6.013,149.051
C06299=1167.394,18.583,-47.297,-179.913,6.012,149.052
C06300=1167.399,18.334,-47.283,-179.915,6.011,149.052
C06301=1167.404,18.084,-47.269,-179.917,6.011,149.053
C06302=1167.409,17.835,-47.255,-179.920,6.010,149.054
C06303=1167.414,17.585,-47.241,-179.922,6.009,149.054
C06304=1167.419,17.335,-47.226,-179.925,6.009,149.055
C06305=1167.424,17.087,-47.212,-179.927,6.008,149.055
C06306=1167.429,16.837,-47.197,-179.930,6.007,149.056
C06307=1167.434,16.588,-47.183,-179.932,6.006,149.056
C06308=1167.439,16.338,-47.169,-179.935,6.006,149.057
C06309=1167.444,16.088,-47.155,-179.938,6.005,149.058
C06310=1167.450,15.839,-47.141,-179.940,6.004,149.058
C06311=1167.455,15.589,-47.126,-179.943,6.004,149.059
C06312=1167.460,15.340,-47.112,-179.945,6.003,149.059
C06313=1167.465,15.090,-47.098,-179.948,6.002,149.060
C06314=1167.470,14.841,-47.084,-179.951,6.001,149.061
C06315=1167.475,14.591,-47.070,-179.953,6.000,149.061
C06316=1167.480,14.341,-47.056,-179.955,6.000,149.062
C06317=1167.485,14.091,-47.042,-179.958,5.999,149.062
C06318=1167.491,13.842,-47.028,-179.960,5.999,149.063
C06319=1167.496,13.592,-47.014,-179.962,5.998,149.063
C06320=1167.501,13.343,-46.999,-179.966,5.996,149.064
C06321=1167.506,13.093,-46.985,-179.968,5.996,149.065
C06322=1167.511,12.844,-46.972,-179.971,5.995,149.065
C06323=1167.516,12.595,-46.957,-179.973,5.995,149.066
C06324=1167.520,12.345,-46.943,-179.975,5.994,149.066
C06325=1167.526,12.096,-46.929,-179.978,5.993,149.067
C06326=1167.531,11.846,-46.916,-179.981,5.993,149.068
C06327=1167.536,11.596,-46.901,-179.983,5.992,149.068
C06328=1167.541,11.346,-46.887,-179.986,5.991,149.069
C06329=1167.547,11.097,-46.873,-179.988,5.990,149.069
C06330=1167.551,10.848,-46.860,-179.991,5.990,149.070
C06331=1167.556,10.598,-46.845,-179.993,5.989,149.071
C06332=1167.562,10.348,-46.832,-179.996,5.988,149.071
C06333=1167.567,10.099,-46.818,-179.998,5.988,149.072
C06334=1167.572,9.849,-46.804,179.999,5.987,149.072
C06335=1167.577,9.600,-46.790,179.997,5.986,149.073
C06336=1167.582,9.350,-46.775,179.995,5.986,149.074
C06337=1167.587,9.100,-46.762,179.991,5.984,149.074
C06338=1167.592,8.851,-46.748,179.989,5.984,149.075
C06339=1167.597,8.602,-46.734,179.987,5.983,149.075
C06340=1167.602,8.352,-46.720,179.984,5.983,149.076
C06341=1167.608,8.102,-46.707,179.982,5.982,149.076
C06342=1167.612,7.853,-46.693,179.979,5.981,149.077
C06343=1167.617,7.603,-46.679,179.976,5.981,149.078
C06344=1167.623,7.353,-46.666,179.974,5.980,149.078
C06345=1167.628,7.104,-46.651,179.972,5.980,149.079
C06346=1167.632,6.854,-46.638,179.969,5.979,149.079
C06347=1167.638,6.605,-46.624,179.967,5.978,149.080
C06348=1167.643,6.355,-46.610,179.964,5.977,149.081
C06349=1167.649,6.106,-46.596,179.961,5.976,149.081
C06350=1167.653,5.857,-46.583,179.959,5.976,149.082
C06351=1167.658,5.606,-46.569,179.957,5.975,149.082
C06352=1167.664,5.357,-46.555,179.954,5.974,149.083
C06353=1167.669,5.107,-46.542,179.951,5.974,149.084
C06354=1167.674,4.858,-46.528,179.949,5.973,149.084
C06355=1167.679,4.609,-46.514,179.946,5.973,149.085
C06356=1167.684,4.358,-46.500,179.944,5.972,149.085
C06357=1167.689,4.109,-46.487,179.942,5.971,149.086
C06358=1167.694,3.860,-46.473,179.939,5.970,149.087
C06359=1167.700,3.610,-46.460,179.937,5.970,149.087
C06360=1167.704,3.361,-46.446,179.934,5.969,149.088
C06361=1167.709,3.110,-46.432,179.931,5.968,149.088
C06362=1167.715,2.861,-46.418,179.929,5.967,149.089
C06363=1167.719,2.611,-46.405,179.927,5.967,149.090
C06364=1167.725,2.343,-46.391,179.924,5.966,149.090
C06365=1167.731,2.073,-46.376,179.921,5.966,149.091
C06366=1167.736,1.804,-46.361,179.919,5.965,149.092
C06367=1167.742,1.534,-46.347,179.915,5.964,149.092
C06368=1167.747,1.285,-46.333,179.913,5.963,149.093
C06369=1167.752,1.035,-46.320,179.911,5.963,149.093
C06370=1167.757,0.786,-46.306,179.908,5.962,149.094
C06371=1167.762,0.536,-46.293,179.906,5.961,149.095
C06372=1167.767,0.287,-46.279,179.903,5.961,149.095
C06373=1167.772,0.037,-46.266,179.901,5.960,149.096
C06374=1167.778,-0.212,-46.252,179.898,5.960,149.096
C06375=1167.783,-0.463,-46.238,179.896,5.959,149.097
C06376=1167.788,-0.711,-46.225,179.893,5.958,149.098
C06377=1167.793,-0.962,-46.212,179.891,5.958,149.098
C06378=1167.798,-1.210,-46.198,179.889,5.957,149.099
C06379=1167.803,-1.461,-46.185,179.886,5.957,149.099
C06380=1167.808,-1.710,-46.172,179.884,5.956,149.100
C06381=1167.813,-1.960,-46.158,179.881,5.955,149.101
C06382=1167.819,-2.209,-46.145,179.878,5.955,149.101
C06383=1167.823,-2.459,-46.131,179.876,5.954,149.102
C06384=1167.829,-2.708,-46.118,179.874,5.954,149.102
C06385=1167.834,-2.958,-46.105,179.871,5.953,149.103
C06386=1167.839,-3.207,-46.091,179.868,5.952,149.104
C06387=1167.844,-3.457,-46.078,179.866,5.951,149.104
C06388=1167.849,-3.707,-46.065,179.863,5.950,149.105
C06389=1167.854,-3.956,-46.051,179.861,5.950,149.105
C06390=1167.860,-4.206,-46.038,179.859,5.949,149.106
C06391=1167.865,-4.455,-46.025,179.856,5.949,149.107
C06392=1167.870,-4.705,-46.011,179.853,5.948,149.107
C06393=1167.875,-4.954,-45.998,179.851,5.947,149.108
C06394=1167.880,-5.205,-45.985,179.848,5.947,149.108
C06395=1167.885,-5.454,-45.972,179.846,5.946,149.109
C06396=1167.890,-5.704,-45.958,179.844,5.946,149.110
C06397=1167.895,-5.953,-45.945,179.841,5.945,149.110
C06398=1167.900,-6.203,-45.932,179.839,5.944,149.111
C06399=1167.906,-6.453,-45.919,179.836,5.944,149.111
C06400=1167.910,-6.701,-45.906,179.834,5.943,149.112
C06401=1167.916,-6.952,-45.892,179.831,5.943,149.113
C06402=1167.921,-7.201,-45.880,179.829,5.942,149.113
C06403=1167.926,-7.451,-45.866,179.826,5.941,149.114
C06404=1167.931,-7.700,-45.853,179.824,5.941,149.114
C06405=1167.936,-7.949,-45.840,179.821,5.940,149.115
C06406=1167.941,-8.200,-45.827,179.819,5.940,149.116
C06407=1167.946,-8.449,-45.814,179.816,5.939,149.116
C06408=1167.952,-8.699,-45.800,179.814,5.938,149.117
C06409=1167.957,-8.949,-45.788,179.811,5.938,149.117
C06410=1167.962,-9.197,-45.775,179.809,5.937,149.118
C06411=1167.967,-9.448,-45.761,179.807,5.937,149.119
C06412=1167.972,-9.697,-45.748,179.804,5.936,149.119
C06413=1167.977,-9.946,-45.736,179.802,5.935,149.120
C06414=1167.982,-10.197,-45.722,179.799,5.935,149.120
C06415=1167.987,-10.446,-45.710,179.796,5.934,149.121
C06416=1167.993,-10.696,-45.696,179.794,5.934,149.122
C06417=1167.998,-10.946,-45.683,179.792,5.933,149.122
C06418=1168.003,-11.194,-45.670,179.789,5.932,149.123
C06419=1168.008,-11.445,-45.657,179.787,5.932,149.123
C06420=1168.013,-11.694,-45.644,179.784,5.931,149.124
C06421=1168.018,-11.943,-45.631,179.782,5.931,149.125
C06422=1168.023,-12.193,-45.618,179.779,5.930,149.125
C06423=1168.029,-12.443,-45.605,179.777,5.929,149.126
C06424=1168.034,-12.692,-45.593,179.774,5.929,149.126
C06425=1168.038,-12.942,-45.580,179.772,5.928,149.127
C06426=1168.044,-13.192,-45.566,179.770,5.928,149.128
C06427=1168.049,-13.441,-45.554,179.767,5.927,149.128
C06428=1168.054,-13.691,-45.541,179.765,5.926,149.129
C06429=1168.059,-13.941,-45.528,179.762,5.926,149.129
C06430=1168.065,-14.190,-45.515,179.759,5.925,149.130
C06431=1168.070,-14.440,-45.502,179.757,5.925,149.131
C06432=1168.074,-14.690,-45.490,179.755,5.924,149.131
C06433=1168.080,-14.939,-45.476,179.752,5.923,149.132
C06434=1168.085,-15.188,-45.464,179.750,5.923,149.132
C06435=1168.090,-15.439,-45.451,179.747,5.922,149.133
C06436=1168.095,-15.688,-45.438,179.745,5.922,149.134
C06437=1168.100,-15.937,-45.426,179.743,5.922,149.134
C06438=1168.106,-16.187,-45.412,179.741,5.921,149.135
C06439=1168.111,-16.437,-45.399,179.738,5.921,149.135
C06440=1168.116,-16.686,-45.387,179.735,5.920,149.136
C06441=1168.121,-16.936,-45.375,179.733,5.919,149.137
C06442=1168.127,-17.186,-45.362,179.731,5.919,149.137
C06443=1168.131,-17.436,-45.349,179.728,5.918,149.138
C06444=1168.137,-17.685,-45.336,179.726,5.918,149.139
C06445=1168.142,-17.934,-45.324,179.723,5.917,149.139
C06446=1168.147,-18.184,-45.311,179.721,5.916,149.140
C06447=1168.151,-18.434,-45.298,179.718,5.916,149.140
C06448=1168.157,-18.683,-45.285,179.716,5.915,149.141
C06449=1168.163,-18.933,-45.273,179.713,5.915,149.142
C06450=1168.168,-19.183,-45.260,179.711,5.914,149.142
C06451=1168.172,-19.433,-45.247,179.709,5.913,149.143
C06452=1168.177,-19.682,-45.235,179.706,5.913,149.143
C06453=1168.183,-19.931,-45.222,179.703,5.913,149.144
C06454=1168.189,-20.181,-45.210,179.701,5.912,149.145
C06455=1168.194,-20.431,-45.197,179.698,5.911,149.145
C06456=1168.198,-20.681,-45.184,179.696,5.911,149.146
C06457=1168.203,-20.930,-45.171,179.694,5.911,149.146
C06458=1168.209,-21.179,-45.159,179.692,5.910,149.147
C06459=1168.214,-21.429,-45.147,179.689,5.910,149.148
C06460=1168.219,-21.679,-45.134,179.687,5.909,149.148
C06461=1168.224,-21.928,-45.122,179.685,5.908,149.149
C06462=1168.229,-22.178,-45.109,179.682,5.908,149.149
C06463=1168.235,-22.428,-45.096,179.679,5.908,149.150
C06464=1168.240,-22.678,-45.084,179.677,5.907,149.151
C06465=1168.245,-22.927,-45.071,179.674,5.906,149.151
C06466=1168.251,-23.177,-45.059,179.672,5.905,149.152
C06467=1168.256,-23.426,-45.047,179.670,5.905,149.152
C06468=1168.261,-23.696,-45.033,179.667,5.905,149.153
C06469=1168.266,-23.966,-45.020,179.664,5.904,149.154
C06470=1168.272,-24.236,-45.006,179.662,5.903,149.154
C06471=1168.278,-24.506,-44.993,179.659,5.903,149.155
C06472=1168.283,-24.755,-44.981,179.657,5.902,149.156
C06473=1168.288,-25.005,-44.968,179.655,5.902,149.156
C06474=1168.293,-25.254,-44.956,179.652,5.901,149.157
C06475=1168.298,-25.505,-44.943,179.649,5.901,149.158
C06476=1168.303,-25.754,-44.930,179.647,5.900,149.158
C06477=1168.308,-26.004,-44.919,179.644,5.899,149.159
C06478=1168.314,-26.253,-44.906,179.642,5.899,149.159
C06479=1168.319,-26.503,-44.894,179.640,5.899,149.160
C06480=1168.324,-26.752,-44.882,179.637,5.899,149.161
C06481=1168.329,-27.002,-44.869,179.635,5.898,149.161
C06482=1168.335,-27.252,-44.857,179.633,5.897,149.162
C06483=1168.339,-27.502,-44.844,179.630,5.897,149.162
C06484=1168.345,-27.752,-44.832,179.628,5.896,149.163
C06485=1168.350,-28.001,-44.820,179.625,5.896,149.164
C06486=1168.355,-28.251,-44.808,179.623,5.895,149.164
C06487=1168.360,-28.500,-44.795,179.620,5.894,149.165
C06488=1168.365,-28.749,-44.782,179.618,5.894,149.165
C06489=1168.371,-28.999,-44.771,179.616,5.894,149.166
C06490=1168.376,-29.249,-44.758,179.613,5.894,149.167
C06491=1168.381,-29.498,-44.747,179.611,5.893,149.167
C06492=1168.386,-29.748,-44.734,179.608,5.892,149.168
C06493=1168.391,-29.998,-44.722,179.606,5.891,149.168
C06494=1168.396,-30.247,-44.710,179.604,5.891,149.169
C06495=1168.402,-30.497,-44.698,179.601,5.891,149.170
C06496=1168.407,-30.747,-44.686,179.599,5.890,149.170
C06497=1168.412,-30.997,-44.673,179.596,5.889,149.171
C06498=1168.417,-31.247,-44.661,179.595,5.889,149.171
C06499=1168.422,-31.496,-44.648,179.592,5.889,149.172
C06500=1168.428,-31.746,-44.637,179.589,5.889,149.173
C06501=1168.432,-31.995,-44.625,179.587,5.888,149.173
C06502=1168.438,-32.245,-44.613,179.584,5.887,149.174
C06503=1168.443,-32.494,-44.600,179.582,5.886,149.174
C06504=1168.448,-32.744,-44.588,179.580,5.886,149.175
C06505=1168.454,-32.994,-44.576,179.577,5.886,149.176
C06506=1168.459,-33.243,-44.564,179.575,5.885,149.176
C06507=1168.463,-33.493,-44.552,179.573,5.885,149.177
C06508=1168.469,-33.743,-44.540,179.570,5.884,149.177
C06509=1168.474,-33.992,-44.528,179.568,5.884,149.178
C06510=1168.479,-34.242,-44.516,179.565,5.883,149.179
C06511=1168.484,-34.492,-44.503,179.563,5.883,149.179
C06512=1168.490,-34.742,-44.492,179.560,5.882,149.180
C06513=1168.495,-34.991,-44.480,179.558,5.881,149.180
C06514=1168.500,-35.240,-44.468,179.556,5.882,149.181
C06515=1168.505,-35.490,-44.456,179.553,5.881,149.182
C06516=1168.511,-35.740,-44.444,179.551,5.881,149.182
C06517=1168.516,-35.990,-44.432,179.549,5.880,149.183
C06518=1168.520,-36.239,-44.420,179.546,5.879,149.184
C06519=1168.526,-36.489,-44.408,179.544,5.879,149.184
C06520=1168.532,-36.738,-44.397,179.541,5.878,149.185
C06521=1168.537,-36.988,-44.384,179.539,5.878,149.185
C06522=1168.542,-37.237,-44.373,179.537,5.878,149.186
C06523=1168.547,-37.487,-44.361,179.535,5.877,149.187
C06524=1168.553,-37.737,-44.349,179.532,5.877,149.187
C06525=1168.558,-37.987,-44.336,179.530,5.876,149.188
C06526=1168.562,-38.236,-44.325,179.527,5.876,149.188
C06527=1168.568,-38.486,-44.313,179.524,5.875,149.189
C06528=1168.573,-38.736,-44.301,179.523,5.875,149.190
C06529=1168.578,-38.986,-44.290,179.520,5.875,149.190
C06530=1168.583,-39.235,-44.277,179.518,5.874,149.191
C06531=1168.588,-39.485,-44.265,179.515,5.873,149.191
C06532=1168.594,-39.735,-44.254,179.513,5.873,149.192
C06533=1168.599,-39.985,-44.242,179.510,5.872,149.193
C06534=1168.605,-40.234,-44.231,179.508,5.872,149.193
C06535=1168.610,-40.483,-44.218,179.506,5.872,149.194
C06536=1168.614,-40.733,-44.207,179.504,5.871,149.195
C06537=1168.620,-40.983,-44.195,179.501,5.871,149.195
C06538=1168.625,-41.233,-44.183,179.499,5.870,149.196
C06539=1168.630,-41.482,-44.172,179.496,5.870,149.196
C06540=1168.635,-41.732,-44.160,179.494,5.869,149.197
C06541=1168.641,-41.982,-44.148,179.492,5.869,149.198
C06542=1168.645,-42.231,-44.136,179.490,5.868,149.198
C06543=1168.651,-42.481,-44.124,179.487,5.868,149.199
C06544=1168.657,-42.730,-44.113,179.484,5.868,149.199
C06545=1168.661,-42.980,-44.101,179.482,5.867,149.200
C06546=1168.667,-43.230,-44.089,179.480,5.867,149.201
C06547=1168.671,-43.479,-44.078,179.478,5.866,149.201
C06548=1168.677,-43.729,-44.066,179.475,5.866,149.202
C06549=1168.682,-43.979,-44.054,179.472,5.866,149.203
C06550=1168.687,-44.229,-44.043,179.470,5.865,149.203
C06551=1168.693,-44.478,-44.032,179.468,5.864,149.204
C06552=1168.698,-44.728,-44.020,179.466,5.864,149.204
C06553=1168.703,-44.978,-44.008,179.463,5.864,149.205
C06554=1168.709,-45.228,-43.997,179.461,5.863,149.205
C06555=1168.713,-45.477,-43.985,179.459,5.863,149.206
C06556=1168.719,-45.727,-43.973,179.456,5.862,149.207
C06557=1168.724,-45.976,-43.962,179.454,5.862,149.207
C06558=1168.729,-46.226,-43.951,179.452,5.862,149.208
C06559=1168.734,-46.476,-43.939,179.449,5.861,149.208
C06560=1168.740,-46.726,-43.927,179.447,5.861,149.209
C06561=1168.744,-46.975,-43.916,179.444,5.860,149.210
C06562=1168.750,-47.224,-43.905,179.442,5.859,149.210
C06563=1168.755,-47.474,-43.893,179.440,5.860,149.211
C06564=1168.760,-47.724,-43.881,179.438,5.859,149.211
C06565=1168.766,-47.974,-43.870,179.435,5.859,149.212
C06566=1168.771,-48.224,-43.858,179.433,5.858,149.213
C06567=1168.777,-48.473,-43.847,179.430,5.857,149.213
C06568=1168.781,-48.722,-43.835,179.428,5.858,149.214
C06569=1168.787,-48.972,-43.824,179.426,5.857,149.215
C06570=1168.791,-49.222,-43.812,179.423,5.856,149.215
C06571=1168.797,-49.473,-43.801,179.421,5.856,149.216
C06572=1168.802,-49.742,-43.789,179.418,5.855,149.216
C06573=1168.808,-50.013,-43.777,179.416,5.855,149.217
C06574=1168.814,-50.283,-43.764,179.413,5.854,149.218
C06575=1168.819,-50.554,-43.752,179.411,5.854,149.218
C06576=1168.825,-50.803,-43.740,179.409,5.854,149.219
C06577=1168.830,-51.053,-43.729,179.406,5.854,149.220
C06578=1168.836,-51.302,-43.717,179.404,5.853,149.220
C06579=1168.841,-51.553,-43.707,179.401,5.852,149.221
C06580=1168.845,-51.802,-43.695,179.400,5.852,149.221
C06581=1168.851,-52.052,-43.684,179.397,5.852,149.222
C06582=1168.856,-52.301,-43.673,179.395,5.851,149.223
C06583=1168.861,-52.551,-43.661,179.392,5.851,149.223
C06584=1168.866,-52.801,-43.650,179.389,5.850,149.224
C06585=1168.872,-53.051,-43.639,179.388,5.850,149.224
C06586=1168.877,-53.300,-43.627,179.385,5.850,149.225
C06587=1168.882,-53.550,-43.616,179.383,5.849,149.226
C06588=1168.887,-53.800,-43.604,179.380,5.849,149.226
C06589=1168.893,-54.049,-43.594,179.379,5.849,149.227
C06590=1168.898,-54.299,-43.583,179.376,5.848,149.227
C06591=1168.903,-54.549,-43.571,179.373,5.848,149.228
C06592=1168.908,-54.798,-43.560,179.371,5.847,149.229
C06593=1168.914,-55.048,-43.549,179.369,5.847,149.229
C06594=1168.919,-55.298,-43.537,179.367,5.847,149.230
C06595=1168.923,-55.548,-43.526,179.364,5.846,149.231
C06596=1168.930,-55.797,-43.515,179.362,5.845,149.231
C06597=1168.934,-56.047,-43.504,179.359,5.845,149.232
C06598=1168.939,-56.297,-43.493,179.357,5.845,149.232
C06599=1168.945,-56.546,-43.481,179.355,5.845,149.233
C06600=1168.950,-56.796,-43.471,179.353,5.844,149.234
C06601=1168.955,-57.046,-43.459,179.350,5.843,149.234
C06602=1168.960,-57.295,-43.448,179.348,5.844,149.235
C06603=1168.966,-57.545,-43.437,179.346,5.843,149.235
C06604=1168.971,-57.795,-43.426,179.343,5.843,149.236
C06605=1168.976,-58.044,-43.416,179.341,5.842,149.236
C06606=1168.982,-58.294,-43.404,179.339,5.842,149.237
C06607=1168.986,-58.544,-43.393,179.336,5.842,149.238
C06608=1168.992,-58.793,-43.382,179.334,5.841,149.238
C06609=1168.997,-59.043,-43.371,179.332,5.841,149.239
C06610=1169.002,-59.293,-43.359,179.330,5.841,149.240
C06611=1169.008,-59.543,-43.349,179.327,5.840,149.240
C06612=1169.012,-59.792,-43.338,179.325,5.839,149.241
C06613=1169.019,-60.042,-43.327,179.323,5.839,149.241
C06614=1169.023,-60.292,-43.316,179.321,5.839,149.242
C06615=1169.028,-60.542,-43.305,179.318,5.839,149.243
C06616=1169.034,-60.791,-43.294,179.316,5.838,149.243
C06617=1169.038,-61.040,-43.283,179.313,5.837,149.244
C06618=1169.044,-61.291,-43.272,179.311,5.838,149.244
C06619=1169.049,-61.540,-43.261,179.309,5.837,149.245
C06620=1169.054,-61.790,-43.250,179.306,5.837,149.246
C06621=1169.060,-62.039,-43.239,179.304,5.836,149.246
C06622=1169.065,-62.290,-43.228,179.302,5.836,149.247
C06623=1169.071,-62.539,-43.217,179.300,5.835,149.247
C06624=1169.076,-62.789,-43.207,179.297,5.835,149.248
C06625=1169.080,-63.038,-43.195,179.295,5.835,149.249
C06626=1169.086,-63.288,-43.185,179.293,5.835,149.249
C06627=1169.091,-63.538,-43.173,179.290,5.834,149.250
C06628=1169.097,-63.788,-43.163,179.288,5.833,149.250
C06629=1169.102,-64.037,-43.152,179.286,5.834,149.251
C06630=1169.107,-64.287,-43.141,179.284,5.833,149.252
C06631=1169.112,-64.536,-43.130,179.281,5.832,149.252
C06632=1169.117,-64.787,-43.120,179.279,5.832,149.253
C06633=1169.123,-65.036,-43.109,179.277,5.832,149.253
C06634=1169.128,-65.286,-43.097,179.275,5.831,149.254
C06635=1169.134,-65.536,-43.087,179.272,5.831,149.255
C06636=1169.138,-65.785,-43.076,179.270,5.830,149.255
C06637=1169.144,-66.035,-43.066,179.268,5.830,149.256
C06638=1169.149,-66.284,-43.054,179.265,5.830,149.257
C06639=1169.154,-66.534,-43.044,179.263,5.829,149.257
C06640=1169.160,-66.784,-43.033,179.261,5.830,149.258
C06641=1169.165,-67.034,-43.022,179.259,5.829,149.258
C06642=1169.170,-67.284,-43.012,179.256,5.828,149.259
C06643=1169.175,-67.534,-43.001,179.254,5.828,149.259
C06644=1169.180,-67.783,-42.990,179.252,5.828,149.260
C06645=1169.185,-68.033,-42.980,179.250,5.827,149.261
C06646=1169.191,-68.283,-42.969,179.247,5.827,149.261
C06647=1169.196,-68.532,-42.958,179.245,5.827,149.262
C06648=1169.201,-68.782,-42.948,179.243,5.826,149.262
C06649=1169.206,-69.032,-42.937,179.240,5.826,149.263
C06650=1169.212,-69.281,-42.926,179.238,5.826,149.264
C06651=1169.217,-69.532,-42.915,179.236,5.826,149.264
C06652=1169.223,-69.781,-42.905,179.234,5.825,149.265
C06653=1169.228,-70.031,-42.894,179.231,5.825,149.266
C06654=1169.233,-70.280,-42.883,179.229,5.824,149.266
C06655=1169.239,-70.530,-42.873,179.227,5.824,149.267
C06656=1169.244,-70.780,-42.863,179.225,5.823,149.267
C06657=1169.249,-71.029,-42.852,179.222,5.824,149.268
C06658=1169.254,-71.279,-42.841,179.220,5.823,149.268
C06659=1169.260,-71.529,-42.831,179.218,5.823,149.269
C06660=1169.265,-71.779,-42.820,179.216,5.823,149.270
C06661=1169.270,-72.028,-42.809,179.213,5.822,149.270
C06662=1169.275,-72.278,-42.799,179.211,5.821,149.271
C06663=1169.281,-72.528,-42.789,179.208,5.821,149.272
C06664=1169.286,-72.778,-42.778,179.207,5.821,149.272
C06665=1169.291,-73.027,-42.767,179.204,5.821,149.273
C06666=1169.297,-73.276,-42.757,179.202,5.820,149.273
C06667=1169.302,-73.527,-42.746,179.200,5.820,149.274
C06668=1169.307,-73.776,-42.736,179.197,5.820,149.275
C06669=1169.312,-74.026,-42.726,179.195,5.819,149.275
C06670=1169.318,-74.276,-42.715,179.193,5.819,149.276
C06671=1169.322,-74.526,-42.704,179.191,5.819,149.276
C06672=1169.328,-74.775,-42.694,179.188,5.818,149.277
C06673=1169.334,-75.025,-42.684,179.187,5.818,149.277
C06674=1169.339,-75.275,-42.673,179.184,5.818,149.278
C06675=1169.344,-75.524,-42.663,179.182,5.817,149.279
C06676=1169.349,-75.796,-42.652,179.179,5.817,149.279
C06677=1169.356,-76.066,-42.640,179.177,5.817,149.280
C06678=1169.361,-76.337,-42.629,179.175,5.816,149.281
C06679=1169.367,-76.609,-42.618,179.172,5.816,149.281
C06680=1169.372,-76.858,-42.607,179.169,5.815,149.282
C06681=1169.377,-77.109,-42.597,179.168,5.815,149.282
C06682=1169.383,-77.358,-42.587,179.165,5.815,149.283
C06683=1169.388,-77.608,-42.576,179.163,5.814,149.284
C06684=1169.393,-77.858,-42.566,179.161,5.815,149.284
C06685=1169.398,-78.107,-42.556,179.159,5.814,149.285
C06686=1169.404,-78.356,-42.545,179.156,5.813,149.286
C06687=1169.409,-78.606,-42.535,179.154,5.813,149.286
C06688=1169.414,-78.856,-42.525,179.152,5.813,149.287
C06689=1169.419,-79.106,-42.514,179.150,5.812,149.287
C06690=1169.425,-79.356,-42.504,179.147,5.813,149.288
C06691=1169.430,-79.605,-42.494,179.145,5.812,149.288
C06692=1169.435,-79.856,-42.483,179.143,5.812,149.289
C06693=1169.440,-80.105,-42.473,179.141,5.812,149.290
C06694=1169.446,-80.354,-42.463,179.138,5.811,149.290
C06695=1169.451,-80.605,-42.453,179.136,5.810,149.291
C06696=1169.456,-80.854,-42.442,179.134,5.811,149.291
C06697=1169.462,-81.104,-42.432,179.132,5.810,149.292
C06698=1169.467,-81.354,-42.422,179.129,5.810,149.293
C06699=1169.472,-81.603,-42.412,179.128,5.810,149.293
C06700=1169.478,-81.853,-42.402,179.125,5.809,149.294
C06701=1169.483,-82.103,-42.391,179.123,5.808,149.294
C06702=1169.488,-82.353,-42.382,179.121,5.809,149.295
C06703=1169.494,-82.603,-42.371,179.118,5.808,149.296
C06704=1169.499,-82.852,-42.362,179.116,5.808,149.296
C06705=1169.504,-83.102,-42.351,179.114,5.808,149.297
C06706=1169.510,-83.352,-42.341,179.112,5.807,149.297
C06707=1169.515,-83.601,-42.331,179.110,5.807,149.298
C06708=1169.519,-83.851,-42.321,179.107,5.807,149.299
C06709=1169.525,-84.101,-42.311,179.105,5.806,149.299
C06710=1169.531,-84.350,-42.300,179.103,5.806,149.300
C06711=1169.536,-84.600,-42.290,179.101,5.806,149.300
C06712=1169.540,-84.850,-42.280,179.098,5.805,149.301
C06713=1169.546,-85.100,-42.271,179.097,5.805,149.302
C06714=1169.552,-85.349,-42.261,179.094,5.805,149.302
C06715=1169.557,-85.600,-42.250,179.092,5.804,149.303
C06716=1169.562,-85.849,-42.240,179.090,5.804,149.303
C06717=1169.567,-86.098,-42.230,179.087,5.804,149.304
C06718=1169.572,-86.349,-42.220,179.086,5.804,149.304
C06719=1169.578,-86.599,-42.210,179.083,5.803,149.305
C06720=1169.583,-86.848,-42.200,179.081,5.803,149.306
C06721=1169.589,-87.098,-42.190,179.079,5.803,149.306
C06722=1169.594,-87.348,-42.180,179.077,5.802,149.307
C06723=1169.599,-87.597,-42.170,179.074,5.802,149.307
C06724=1169.604,-87.847,-42.160,179.072,5.802,149.308
C06725=1169.610,-88.097,-42.150,179.070,5.801,149.309
C06726=1169.614,-88.347,-42.140,179.068,5.801,149.309
C06727=1169.620,-88.596,-42.130,179.065,5.801,149.310
C06728=1169.626,-88.846,-42.120,179.063,5.800,149.310
C06729=1169.631,-89.096,-42.111,179.061,5.801,149.311
C06730=1169.636,-89.345,-42.101,179.059,5.800,149.312
C06731=1169.641,-89.595,-42.090,179.056,5.800,149.312
C06732=1169.646,-89.845,-42.081,179.055,5.800,149.313
C06733=1169.652,-90.095,-42.071,179.052,5.799,149.313
C06734=1169.658,-90.344,-42.061,179.050,5.799,149.314
C06735=1169.663,-90.594,-42.051,179.048,5.798,149.314
C06736=1169.668,-90.844,-42.041,179.046,5.798,149.315
C06737=1169.673,-91.094,-42.031,179.044,5.798,149.316
C06738=1169.678,-91.343,-42.022,179.041,5.798,149.316
C06739=1169.684,-91.593,-42.011,179.039,5.797,149.317
C06740=1169.689,-91.843,-42.003,179.037,5.797,149.318
C06741=1169.694,-92.093,-41.992,179.035,5.796,149.318
C06742=1169.700,-92.342,-41.982,179.033,5.797,149.319
C06743=1169.705,-92.592,-41.973,179.031,5.796,149.319
C06744=1169.710,-92.842,-41.963,179.028,5.796,149.320
C06745=1169.715,-93.091,-41.953,179.026,5.796,149.320
C06746=1169.721,-93.342,-41.943,179.024,5.795,149.321
C06747=1169.726,-93.591,-41.933,179.022,5.795,149.322
C06748=1169.731,-93.841,-41.923,179.020,5.795,149.322
C06749=1169.737,-94.091,-41.914,179.017,5.794,149.323
C06750=1169.742,-94.340,-41.904,179.016,5.794,149.323
C06751=1169.748,-94.590,-41.895,179.013,5.794,149.324
C06752=1169.753,-94.839,-41.885,179.011,5.794,149.324
C06753=1169.758,-95.090,-41.875,179.009,5.793,149.325
C06754=1169.763,-95.340,-41.865,179.006,5.793,149.326
C06755=1169.768,-95.589,-41.856,179.004,5.793,149.326
C06756=1169.774,-95.839,-41.846,179.002,5.792,149.327
C06757=1169.779,-96.089,-41.836,179.001,5.792,149.327
C06758=1169.785,-96.339,-41.827,178.998,5.792,149.328
C06759=1169.790,-96.588,-41.817,178.996,5.791,149.329
C06760=1169.795,-96.837,-41.807,178.994,5.792,149.329
C06761=1169.800,-97.088,-41.798,178.991,5.791,149.330
C06762=1169.806,-97.338,-41.788,178.989,5.791,149.330
C06763=1169.811,-97.587,-41.779,178.987,5.790,149.331
C06764=1169.816,-97.837,-41.769,178.984,5.790,149.332
C06765=1169.822,-98.087,-41.760,178.983,5.790,149.332
C06766=1169.827,-98.336,-41.749,178.981,5.789,149.333
C06767=1169.832,-98.586,-41.741,178.979,5.790,149.333
C06768=1169.838,-98.836,-41.730,178.976,5.789,149.334
C06769=1169.843,-99.086,-41.721,178.974,5.789,149.334
C06770=1169.849,-99.335,-41.711,178.972,5.789,149.335
C06771=1169.853,-99.586,-41.702,178.969,5.788,149.336
C06772=1169.859,-99.835,-41.692,178.968,5.788,149.336
C06773=1169.864,-100.085,-41.683,178.966,5.787,149.337
C06774=1169.870,-100.335,-41.673,178.964,5.788,149.337
C06775=1169.875,-100.584,-41.664,178.961,5.787,149.338
C06776=1169.880,-100.834,-41.655,178.959,5.787,149.339
C06777=1169.886,-101.084,-41.645,178.957,5.787,149.339
C06778=1169.891,-101.334,-41.636,178.954,5.786,149.340
C06779=1169.896,-101.583,-41.625,178.953,5.786,149.340
C06780=1169.902,-101.855,-41.615,178.950,5.786,149.341
C06781=1169.907,-102.127,-41.605,178.948,5.785,149.341
C06782=1169.913,-102.399,-41.595,178.946,5.786,149.342
C06783=1169.920,-102.671,-41.584,178.943,5.785,149.343
C06784=1169.925,-102.920,-41.575,178.941,5.784,149.343
C06785=1169.930,-103.170,-41.566,178.939,5.784,149.344
C06786=1169.936,-103.420,-41.556,178.937,5.784,149.345
C06787=1169.941,-103.670,-41.547,178.935,5.784,149.345
C06788=1169.946,-103.919,-41.537,178.932,5.784,149.346
C06789=1169.951,-104.170,-41.528,178.931,5.784,149.346
C06790=1169.956,-104.420,-41.519,178.929,5.783,149.347
C06791=1169.962,-104.669,-41.509,178.926,5.783,149.347
C06792=1169.967,-104.919,-41.500,178.924,5.783,149.348
C06793=1169.972,-105.169,-41.491,178.922,5.782,149.349
C06794=1169.978,-105.418,-41.481,178.920,5.782,149.349
C06795=1169.983,-105.668,-41.472,178.918,5.782,149.350
C06796=1169.988,-105.918,-41.463,178.916,5.782,149.350
C06797=1169.994,-106.168,-41.453,178.914,5.781,149.351
C06798=1169.999,-106.418,-41.444,178.912,5.782,149.352
C06799=1170.004,-106.667,-41.435,178.909,5.781,149.352
C06800=1170.009,-106.917,-41.425,178.907,5.780,149.353
C06801=1170.015,-107.167,-41.416,178.905,5.780,149.353
C06802=1170.020,-107.417,-41.407,178.903,5.780,149.354
C06803=1170.026,-107.667,-41.398,178.901,5.780,149.354
C06804=1170.031,-107.916,-41.388,178.899,5.779,149.355
C06805=1170.036,-108.166,-41.379,178.897,5.779,149.355
C06806=1170.042,-108.416,-41.370,178.894,5.779,149.356
C06807=1170.047,-108.665,-41.361,178.893,5.779,149.357
C06808=1170.052,-108.914,-41.351,178.890,5.779,149.357
C06809=1170.057,-109.164,-41.343,178.888,5.778,149.358
C06810=1170.063,-109.414,-41.333,178.886,5.778,149.358
C06811=1170.068,-109.664,-41.324,178.884,5.777,149.359
C06812=1170.074,-109.914,-41.315,178.882,5.778,149.359
C06813=1170.079,-110.163,-41.306,178.879,5.777,149.360
C06814=1170.084,-110.414,-41.296,178.878,5.777,149.361
C06815=1170.090,-110.663,-41.287,178.876,5.776,149.361
C06816=1170.095,-110.913,-41.278,178.874,5.777,149.362
C06817=1170.100,-111.163,-41.269,178.871,5.776,149.362
C06818=1170.106,-111.413,-41.259,178.870,5.776,149.363
C06819=1170.111,-111.662,-41.250,178.867,5.776,149.364
C06820=1170.116,-111.912,-41.241,178.865,5.776,149.364
C06821=1170.121,-112.162,-41.233,178.863,5.775,149.365
C06822=1170.127,-112.412,-41.223,178.861,5.775,149.365
C06823=1170.132,-112.662,-41.214,178.859,5.775,149.366
C06824=1170.138,-112.911,-41.206,178.856,5.774,149.366
C06825=1170.143,-113.161,-41.197,178.855,5.774,149.367
C06826=1170.148,-113.410,-41.187,178.853,5.773,149.367
C06827=1170.154,-113.661,-41.178,178.850,5.774,149.368
C06828=1170.159,-113.910,-41.169,178.848,5.773,149.369
C06829=1170.164,-114.160,-41.160,178.846,5.774,149.369
C06830=1170.169,-114.410,-41.151,178.844,5.773,149.370
C06831=1170.174,-114.660,-41.142,178.842,5.773,149.370
C06832=1170.180,-114.910,-41.133,178.840,5.772,149.371
C06833=1170.186,-115.159,-41.124,178.838,5.772,149.372
C06834=1170.191,-115.409,-41.115,178.836,5.772,149.372
C06835=1170.196,-115.659,-41.106,178.834,5.772,149.373
C06836=1170.202,-115.909,-41.097,178.832,5.771,149.373
C06837=1170.207,-116.159,-41.088,178.830,5.771,149.374
C06838=1170.213,-116.409,-41.079,178.827,5.771,149.374
C06839=1170.218,-116.659,-41.070,178.826,5.771,149.375
C06840=1170.223,-116.909,-41.061,178.824,5.770,149.375
C06841=1170.228,-117.157,-41.052,178.821,5.770,149.376
C06842=1170.234,-117.407,-41.043,178.819,5.770,149.377
C06843=1170.239,-117.657,-41.034,178.817,5.770,149.377
C06844=1170.244,-117.907,-41.025,178.815,5.770,149.378
C06845=1170.250,-118.157,-41.016,178.813,5.769,149.378
C06846=1170.255,-118.407,-41.007,178.811,5.769,149.379
C06847=1170.261,-118.656,-40.999,178.809,5.768,149.379
C06848=1170.266,-118.906,-40.990,178.807,5.768,149.380
C06849=1170.271,-119.156,-40.981,178.804,5.768,149.381
C06850=1170.277,-119.406,-40.972,178.803,5.768,149.381
C06851=1170.282,-119.656,-40.963,178.800,5.767,149.382
C06852=1170.287,-119.906,-40.954,178.798,5.768,149.382
C06853=1170.293,-120.155,-40.946,178.796,5.767,149.383
C06854=1170.298,-120.405,-40.937,178.795,5.767,149.383
C06855=1170.303,-120.655,-40.928,178.792,5.767,149.384
C06856=1170.308,-120.904,-40.919,178.790,5.767,149.385
C06857=1170.313,-121.154,-40.910,178.788,5.766,149.385
C06858=1170.319,-121.404,-40.901,178.786,5.766,149.386
C06859=1170.325,-121.654,-40.892,178.784,5.766,149.386
C06860=1170.330,-121.903,-40.883,178.782,5.766,149.387
C06861=1170.335,-122.153,-40.875,178.780,5.765,149.387
C06862=1170.341,-122.404,-40.866,178.778,5.765,149.388
C06863=1170.346,-122.654,-40.857,178.776,5.765,149.388
C06864=1170.352,-122.903,-40.849,178.774,5.765,149.389
C06865=1170.357,-123.153,-40.840,178.771,5.764,149.390
C06866=1170.362,-123.402,-40.831,178.770,5.764,149.390
C06867=1170.367,-123.652,-40.822,178.767,5.764,149.391
C06868=1170.373,-123.901,-40.814,178.766,5.764,149.391
C06869=1170.379,-124.152,-40.806,178.763,5.763,149.392
C06870=1170.384,-124.402,-40.797,178.762,5.763,149.392
C06871=1170.389,-124.652,-40.788,178.759,5.763,149.393
C06872=1170.394,-124.901,-40.779,178.758,5.763,149.393
C06873=1170.400,-125.151,-40.770,178.755,5.762,149.394
C06874=1170.405,-125.400,-40.761,178.753,5.762,149.395
C06875=1170.410,-125.651,-40.753,178.751,5.762,149.395
C06876=1170.416,-125.901,-40.744,178.749,5.762,149.396
C06877=1170.421,-126.150,-40.736,178.747,5.761,149.396
C06878=1170.427,-126.400,-40.727,178.745,5.761,149.397
C06879=1170.432,-126.650,-40.719,178.743,5.761,149.397
C06880=1170.438,-126.899,-40.710,178.741,5.761,149.398
C06881=1170.442,-127.149,-40.702,178.739,5.760,149.399
C06882=1170.447,-127.399,-40.693,178.737,5.760,149.399
C06883=1170.453,-127.649,-40.684,178.736,5.760,149.400
C06884=1170.032,-127.660,-40.725,178.732,5.764,149.401
C06885=1170.027,-127.410,-40.734,178.733,5.764,149.401
C06886=1170.021,-127.160,-40.743,178.735,5.764,149.400
C06887=1170.015,-126.910,-40.751,178.738,5.764,149.400
C06888=1170.010,-126.660,-40.760,178.740,5.765,149.399
C06889=1170.005,-126.411,-40.769,178.741,5.765,149.399
C06890=1170.000,-126.161,-40.778,178.744,5.765,149.398
C06891=1169.994,-125.911,-40.785,178.746,5.765,149.397
C06892=1169.989,-125.661,-40.794,178.748,5.766,149.397
C06893=1169.984,-125.412,-40.803,178.749,5.766,149.397
C06894=1169.979,-125.162,-40.811,178.752,5.766,149.396
C06895=1169.973,-124.913,-40.820,178.754,5.766,149.395
C06896=1169.968,-124.663,-40.829,178.756,5.767,149.395
C06897=1169.963,-124.412,-40.837,178.758,5.766,149.394
C06898=1169.957,-124.162,-40.846,178.760,5.767,149.394
C06899=1169.952,-123.913,-40.854,178.762,5.767,149.393
C06900=1169.946,-123.663,-40.863,178.764,5.768,149.393
C06901=1169.941,-123.414,-40.872,178.766,5.767,149.392
C06902=1169.936,-123.164,-40.881,178.768,5.768,149.391
C06903=1169.930,-122.914,-40.889,178.770,5.768,149.391
C06904=1169.925,-122.664,-40.898,178.772,5.769,149.390
C06905=1169.920,-122.414,-40.907,178.774,5.769,149.390
C06906=1169.914,-122.164,-40.916,178.776,5.769,149.389
C06907=1169.909,-121.914,-40.925,178.778,5.769,149.389
C06908=1169.903,-121.665,-40.934,178.781,5.770,149.388
C06909=1169.898,-121.415,-40.943,178.782,5.770,149.388
C06910=1169.893,-121.165,-40.951,178.785,5.770,149.387
C06911=1169.887,-120.916,-40.960,178.786,5.770,149.386
C06912=1169.882,-120.665,-40.969,178.789,5.771,149.386
C06913=1169.876,-120.416,-40.977,178.791,5.770,149.385
C06914=1169.871,-120.166,-40.986,178.793,5.771,149.385
C06915=1169.866,-119.916,-40.995,178.794,5.771,149.384
C06916=1169.861,-119.666,-41.004,178.797,5.771,149.383
C06917=1169.856,-119.417,-41.013,178.799,5.771,149.383
C06918=1169.850,-119.167,-41.022,178.801,5.772,149.382
C06919=1169.845,-118.918,-41.030,178.803,5.772,149.382
C06920=1169.839,-118.668,-41.039,178.805,5.772,149.381
C06921=1169.834,-118.418,-41.048,178.807,5.772,149.381
C06922=1169.828,-118.168,-41.057,178.810,5.773,149.380
C06923=1169.823,-117.918,-41.066,178.811,5.773,149.380
C06924=1169.818,-117.668,-41.075,178.813,5.774,149.379
C06925=1169.812,-117.419,-41.084,178.815,5.773,149.378
C06926=1169.807,-117.169,-41.093,178.818,5.774,149.378
C06927=1169.802,-116.919,-41.102,178.819,5.774,149.377
C06928=1169.797,-116.669,-41.110,178.822,5.774,149.377
C06929=1169.792,-116.419,-41.119,178.823,5.774,149.376
C06930=1169.786,-116.169,-41.129,178.826,5.775,149.376
C06931=1169.780,-115.919,-41.138,178.828,5.775,149.375
C06932=1169.775,-115.670,-41.147,178.830,5.775,149.375
C06933=1169.770,-115.420,-41.155,178.832,5.775,149.374
C06934=1169.764,-115.171,-41.164,178.834,5.776,149.373
C06935=1169.759,-114.921,-41.173,178.836,5.776,149.373
C06936=1169.753,-114.671,-41.182,178.838,5.776,149.372
C06937=1169.748,-114.421,-41.191,178.841,5.777,149.372
C06938=1169.743,-114.171,-41.201,178.842,5.777,149.371
C06939=1169.738,-113.922,-41.210,178.845,5.777,149.370
C06940=1169.733,-113.672,-41.219,178.847,5.777,149.370
C06941=1169.726,-113.422,-41.228,178.849,5.778,149.369
C06942=1169.721,-113.172,-41.237,178.851,5.777,149.369
C06943=1169.716,-112.923,-41.246,178.853,5.778,149.368
C06944=1169.711,-112.673,-41.255,178.855,5.778,149.368
C06945=1169.706,-112.423,-41.263,178.857,5.779,149.367
C06946=1169.700,-112.173,-41.273,178.859,5.779,149.367
C06947=1169.695,-111.924,-41.283,178.862,5.779,149.366
C06948=1169.690,-111.674,-41.291,178.863,5.779,149.365
C06949=1169.685,-111.424,-41.300,178.865,5.780,149.365
C06950=1169.679,-111.174,-41.310,178.867,5.779,149.364
C06951=1169.674,-110.924,-41.319,178.870,5.780,149.364
C06952=1169.668,-110.674,-41.328,178.872,5.781,149.363
C06953=1169.663,-110.425,-41.337,178.874,5.780,149.363
C06954=1169.657,-110.175,-41.346,178.876,5.781,149.362
C06955=1169.652,-109.925,-41.355,178.878,5.781,149.361
C06956=1169.647,-109.676,-41.364,178.880,5.781,149.361
C06957=1169.642,-109.426,-41.373,178.882,5.781,149.360
C06958=1169.636,-109.176,-41.383,178.885,5.782,149.360
C06959=1169.631,-108.926,-41.392,178.886,5.782,149.359
C06960=1169.626,-108.676,-41.401,178.889,5.782,149.358
C06961=1169.621,-108.427,-41.410,178.891,5.782,149.358
C06962=1169.615,-108.176,-41.419,178.893,5.783,149.357
C06963=1169.610,-107.927,-41.429,178.895,5.783,149.357
C06964=1169.605,-107.677,-41.438,178.897,5.783,149.356
C06965=1169.599,-107.427,-41.448,178.899,5.784,149.356
C06966=1169.594,-107.177,-41.456,178.901,5.784,149.355
C06967=1169.589,-106.928,-41.466,178.903,5.784,149.355
C06968=1169.583,-106.678,-41.476,178.906,5.784,149.354
C06969=1169.578,-106.428,-41.484,178.908,5.785,149.353
C06970=1169.573,-106.179,-41.494,178.909,5.785,149.353
C06971=1169.567,-105.929,-41.504,178.912,5.785,149.352
C06972=1169.562,-105.679,-41.512,178.914,5.786,149.352
C06973=1169.556,-105.429,-41.521,178.916,5.785,149.351
C06974=1169.551,-105.179,-41.532,178.918,5.786,149.350
C06975=1169.546,-104.930,-41.540,178.920,5.786,149.350
C06976=1169.541,-104.680,-41.549,178.923,5.787,149.349
C06977=1169.535,-104.430,-41.560,178.924,5.787,149.349
C06978=1169.530,-104.180,-41.568,178.927,5.787,149.348
C06979=1169.525,-103.930,-41.577,178.929,5.787,149.348
C06980=1169.519,-103.681,-41.588,178.931,5.788,149.347
C06981=1169.514,-103.431,-41.596,178.933,5.788,149.346
C06982=1169.509,-103.182,-41.606,178.935,5.788,149.346
C06983=1169.503,-102.932,-41.616,178.938,5.788,149.345
C06984=1169.498,-102.682,-41.624,178.939,5.788,149.345
C06985=1169.492,-102.410,-41.635,178.942,5.789,149.344
C06986=1169.486,-102.138,-41.645,178.944,5.790,149.344
C06987=1169.481,-101.866,-41.656,178.946,5.789,149.343
C06988=1169.475,-101.595,-41.666,178.949,5.790,149.342
C06989=1169.470,-101.344,-41.676,178.951,5.790,149.342
C06990=1169.464,-101.094,-41.685,178.953,5.790,149.341
C06991=1169.460,-100.845,-41.695,178.955,5.791,149.340
C06992=1169.454,-100.595,-41.704,178.957,5.791,149.340
C06993=1169.449,-100.346,-41.714,178.960,5.791,149.339
C06994=1169.443,-100.096,-41.723,178.962,5.792,149.339
C06995=1169.438,-99.846,-41.732,178.964,5.791,149.338
C06996=1169.432,-99.596,-41.742,178.966,5.792,149.338
C06997=1169.427,-99.346,-41.751,178.968,5.792,149.337
C06998=1169.421,-99.097,-41.761,178.970,5.793,149.336
C06999=1169.416,-98.847,-41.770,178.972,5.793,149.336
C07000=1169.411,-98.597,-41.781,178.975,5.793,149.335
C07001=1169.405,-98.348,-41.789,178.977,5.794,149.335
C07002=1169.401,-98.098,-41.799,178.979,5.793,149.334
C07003=1169.395,-97.848,-41.809,178.981,5.794,149.333
C07004=1169.390,-97.598,-41.819,178.983,5.794,149.333
C07005=1169.385,-97.348,-41.828,178.985,5.794,149.332
C07006=1169.379,-97.099,-41.838,178.988,5.795,149.332
C07007=1169.374,-96.849,-41.847,178.990,5.795,149.331
C07008=1169.368,-96.599,-41.857,178.992,5.796,149.331
C07009=1169.363,-96.350,-41.867,178.994,5.795,149.330
C07010=1169.357,-96.100,-41.876,178.996,5.796,149.329
C07011=1169.353,-95.850,-41.886,178.999,5.796,149.329
C07012=1169.347,-95.600,-41.896,179.000,5.796,149.328
C07013=1169.342,-95.350,-41.906,179.003,5.797,149.328
C07014=1169.336,-95.100,-41.915,179.005,5.797,149.327
C07015=1169.332,-94.851,-41.925,179.007,5.797,149.327
C07016=1169.326,-94.602,-41.935,179.010,5.798,149.326
C07017=1169.321,-94.352,-41.944,179.011,5.798,149.325
C07018=1169.316,-94.101,-41.954,179.014,5.798,149.325
C07019=1169.310,-93.851,-41.964,179.015,5.798,149.324
C07020=1169.305,-93.602,-41.973,179.018,5.799,149.323
C07021=1169.299,-93.353,-41.984,179.020,5.799,149.323
C07022=1169.294,-93.103,-41.993,179.022,5.799,149.322
C07023=1169.289,-92.853,-42.003,179.025,5.800,149.322
C07024=1169.284,-92.604,-42.012,179.026,5.800,149.321
C07025=1169.279,-92.353,-42.022,179.029,5.800,149.321
C07026=1169.273,-92.103,-42.032,179.031,5.801,149.320
C07027=1169.268,-91.854,-42.042,179.033,5.800,149.319
C07028=1169.262,-91.604,-42.052,179.035,5.801,149.319
C07029=1169.257,-91.355,-42.062,179.037,5.801,149.318
C07030=1169.252,-91.105,-42.072,179.040,5.802,149.318
C07031=1169.246,-90.854,-42.081,179.042,5.802,149.317
C07032=1169.242,-90.605,-42.091,179.044,5.802,149.316
C07033=1169.236,-90.356,-42.101,179.046,5.803,149.316
C07034=1169.230,-90.106,-42.111,179.049,5.803,149.315
C07035=1169.226,-89.856,-42.121,179.050,5.803,149.315
C07036=1169.220,-89.606,-42.131,179.053,5.804,149.314
C07037=1169.215,-89.356,-42.141,179.055,5.804,149.314
C07038=1169.209,-89.107,-42.150,179.057,5.804,149.313
C07039=1169.204,-88.857,-42.160,179.059,5.805,149.312
C07040=1169.199,-88.607,-42.171,179.062,5.804,149.312
C07041=1169.194,-88.358,-42.180,179.064,5.805,149.311
C07042=1169.188,-88.108,-42.190,179.066,5.805,149.311
C07043=1169.182,-87.858,-42.200,179.068,5.805,149.310
C07044=1169.178,-87.608,-42.210,179.071,5.806,149.309
C07045=1169.173,-87.358,-42.220,179.072,5.806,149.309
C07046=1169.167,-87.109,-42.230,179.075,5.806,149.308
C07047=1169.162,-86.859,-42.239,179.077,5.807,149.308
C07048=1169.157,-86.609,-42.250,179.079,5.807,149.307
C07049=1169.151,-86.359,-42.260,179.081,5.807,149.306
C07050=1169.146,-86.110,-42.270,179.084,5.808,149.306
C07051=1169.141,-85.860,-42.280,179.086,5.808,149.305
C07052=1169.136,-85.610,-42.290,179.088,5.809,149.305
C07053=1169.130,-85.361,-42.301,179.090,5.808,149.304
C07054=1169.125,-85.111,-42.310,179.092,5.809,149.304
C07055=1169.120,-84.861,-42.320,179.095,5.809,149.303
C07056=1169.114,-84.611,-42.330,179.096,5.809,149.302
C07057=1169.109,-84.362,-42.341,179.099,5.810,149.302
C07058=1169.104,-84.112,-42.350,179.101,5.810,149.301
C07059=1169.099,-83.862,-42.361,179.103,5.810,149.300
C07060=1169.093,-83.612,-42.371,179.106,5.811,149.300
C07061=1169.088,-83.363,-42.381,179.108,5.811,149.299
C07062=1169.083,-83.112,-42.390,179.110,5.811,149.299
C07063=1169.078,-82.863,-42.401,179.113,5.812,149.298
C07064=1169.072,-82.613,-42.411,179.115,5.812,149.298
C07065=1169.067,-82.363,-42.421,179.117,5.812,149.297
C07066=1169.061,-82.114,-42.432,179.119,5.813,149.296
C07067=1169.057,-81.864,-42.441,179.121,5.812,149.296
C07068=1169.051,-81.615,-42.451,179.123,5.813,149.295
C07069=1169.046,-81.364,-42.462,179.126,5.814,149.295
C07070=1169.040,-81.115,-42.472,179.127,5.814,149.294
C07071=1169.035,-80.865,-42.482,179.130,5.814,149.293
C07072=1169.030,-80.615,-42.493,179.132,5.815,149.293
C07073=1169.025,-80.366,-42.503,179.134,5.814,149.292
C07074=1169.019,-80.116,-42.513,179.137,5.815,149.292
C07075=1169.014,-79.866,-42.523,179.139,5.815,149.291
C07076=1169.009,-79.617,-42.534,179.141,5.815,149.290
C07077=1169.003,-79.367,-42.544,179.144,5.816,149.290
C07078=1168.998,-79.117,-42.554,179.146,5.817,149.289
C07079=1168.993,-78.868,-42.564,179.148,5.816,149.289
C07080=1168.988,-78.617,-42.575,179.150,5.817,149.288
C07081=1168.983,-78.368,-42.585,179.153,5.817,149.287
C07082=1168.977,-78.118,-42.595,179.154,5.817,149.287
C07083=1168.972,-77.868,-42.606,179.157,5.818,149.286
C07084=1168.966,-77.618,-42.616,179.159,5.819,149.286
C07085=1168.961,-77.369,-42.626,179.161,5.818,149.285
C07086=1168.956,-77.119,-42.637,179.163,5.819,149.285
C07087=1168.951,-76.870,-42.647,179.166,5.819,149.284
C07088=1168.945,-76.620,-42.658,179.168,5.819,149.283
C07089=1168.940,-76.349,-42.669,179.170,5.820,149.283
C07090=1168.934,-76.077,-42.680,179.173,5.820,149.282
C07091=1168.928,-75.807,-42.691,179.175,5.821,149.281
C07092=1168.922,-75.535,-42.702,179.178,5.821,149.281
C07093=1168.917,-75.285,-42.713,179.180,5.821,149.280
C07094=1168.912,-75.036,-42.724,179.182,5.822,149.280
C07095=1168.906,-74.786,-42.734,179.185,5.822,149.279
C07096=1168.901,-74.536,-42.745,179.186,5.822,149.278
C07097=1168.896,-74.287,-42.755,179.189,5.823,149.278
C07098=1168.891,-74.036,-42.765,179.191,5.823,149.277
C07099=1168.885,-73.787,-42.776,179.193,5.823,149.276
C07100=1168.880,-73.538,-42.786,179.196,5.824,149.276
C07101=1168.875,-73.288,-42.797,179.198,5.824,149.275
C07102=1168.869,-73.038,-42.807,179.200,5.824,149.275
C07103=1168.864,-72.788,-42.818,179.202,5.824,149.274
C07104=1168.859,-72.538,-42.828,179.205,5.825,149.274
C07105=1168.854,-72.289,-42.839,179.207,5.826,149.273
C07106=1168.848,-72.039,-42.850,179.209,5.826,149.272
C07107=1168.843,-71.790,-42.860,179.212,5.826,149.272
C07108=1168.838,-71.539,-42.870,179.214,5.827,149.271
C07109=1168.832,-71.290,-42.881,179.216,5.826,149.271
C07110=1168.827,-71.040,-42.892,179.218,5.827,149.270
C07111=1168.822,-70.791,-42.902,179.221,5.828,149.269
C07112=1168.817,-70.540,-42.913,179.222,5.828,149.269
C07113=1168.812,-70.291,-42.923,179.225,5.828,149.268
C07114=1168.807,-70.041,-42.934,179.227,5.829,149.268
C07115=1168.801,-69.792,-42.944,179.230,5.829,149.267
C07116=1168.796,-69.541,-42.955,179.232,5.829,149.266
C07117=1168.791,-69.293,-42.966,179.234,5.830,149.266
C07118=1168.786,-69.042,-42.976,179.237,5.830,149.265
C07119=1168.780,-68.793,-42.987,179.238,5.830,149.265
C07120=1168.775,-68.543,-42.998,179.241,5.830,149.264
C07121=1168.770,-68.294,-43.008,179.243,5.831,149.263
C07122=1168.765,-68.043,-43.019,179.245,5.831,149.263
C07123=1168.759,-67.794,-43.030,179.248,5.832,149.262
C07124=1168.754,-67.544,-43.041,179.250,5.832,149.261
C07125=1168.748,-67.294,-43.051,179.252,5.833,149.261
C07126=1168.743,-67.045,-43.062,179.254,5.832,149.260
C07127=1168.738,-66.795,-43.072,179.257,5.833,149.260
C07128=1168.733,-66.545,-43.083,179.259,5.834,149.259
C07129=1168.728,-66.296,-43.094,179.261,5.834,149.259
C07130=1168.723,-66.046,-43.105,179.264,5.834,149.258
C07131=1168.717,-65.797,-43.115,179.266,5.834,149.257
C07132=1168.712,-65.546,-43.127,179.268,5.835,149.257
C07133=1168.706,-65.297,-43.137,179.270,5.835,149.256
C07134=1168.701,-65.047,-43.148,179.273,5.836,149.256
C07135=1168.696,-64.797,-43.159,179.275,5.836,149.255
C07136=1168.691,-64.548,-43.170,179.278,5.837,149.254
C07137=1168.686,-64.298,-43.180,179.280,5.836,149.254
C07138=1168.681,-64.049,-43.191,179.282,5.837,149.253
C07139=1168.675,-63.798,-43.202,179.284,5.838,149.252
C07140=1168.670,-63.549,-43.213,179.286,5.838,149.252
C07141=1168.665,-63.299,-43.224,179.289,5.838,149.251
C07142=1168.659,-63.050,-43.235,179.291,5.839,149.251
C07143=1168.654,-62.800,-43.245,179.294,5.839,149.250
C07144=1168.649,-62.550,-43.257,179.296,5.839,149.249
C07145=1168.643,-62.300,-43.267,179.298,5.840,149.249
C07146=1168.639,-62.051,-43.279,179.301,5.840,149.248
C07147=1168.633,-61.801,-43.289,179.303,5.841,149.248
C07148=1168.628,-61.552,-43.300,179.305,5.840,149.247
C07149=1168.623,-61.301,-43.311,179.307,5.841,149.247
C07150=1168.617,-61.052,-43.322,179.310,5.842,149.246
C07151=1168.612,-60.802,-43.333,179.312,5.842,149.245
C07152=1168.607,-60.553,-43.344,179.314,5.842,149.245
C07153=1168.601,-60.302,-43.355,179.316,5.843,149.244
C07154=1168.597,-60.053,-43.366,179.319,5.843,149.243
C07155=1168.591,-59.803,-43.376,179.321,5.844,149.243
C07156=1168.586,-59.554,-43.388,179.323,5.844,149.242
C07157=1168.581,-59.304,-43.400,179.326,5.844,149.242
C07158=1168.575,-59.054,-43.410,179.328,5.845,149.241
C07159=1168.571,-58.804,-43.421,179.331,5.845,149.240
C07160=1168.566,-58.554,-43.432,179.332,5.845,149.240
C07161=1168.560,-58.305,-43.443,179.335,5.846,149.239
C07162=1168.555,-58.055,-43.454,179.337,5.847,149.239
C07163=1168.549,-57.806,-43.465,179.340,5.847,149.238
C07164=1168.544,-57.556,-43.477,179.342,5.847,149.237
C07165=1168.539,-57.306,-43.488,179.344,5.847,149.237
C07166=1168.534,-57.057,-43.498,179.347,5.848,149.236
C07167=1168.529,-56.807,-43.509,179.349,5.849,149.236
C07168=1168.523,-56.557,-43.521,179.351,5.848,149.235
C07169=1168.518,-56.308,-43.531,179.353,5.849,149.235
C07170=1168.513,-56.058,-43.543,179.356,5.849,149.234
C07171=1168.508,-55.808,-43.555,179.358,5.850,149.233
C07172=1168.503,-55.558,-43.565,179.360,5.850,149.233
C07173=1168.497,-55.309,-43.576,179.363,5.850,149.232
C07174=1168.492,-55.059,-43.588,179.365,5.851,149.231
C07175=1168.487,-54.809,-43.599,179.367,5.851,149.231
C07176=1168.482,-54.560,-43.610,179.370,5.852,149.230
C07177=1168.476,-54.310,-43.621,179.372,5.852,149.230
C07178=1168.472,-54.060,-43.633,179.374,5.853,149.229
C07179=1168.466,-53.811,-43.644,179.377,5.853,149.228
C07180=1168.461,-53.561,-43.655,179.379,5.853,149.228
C07181=1168.456,-53.311,-43.666,179.381,5.853,149.227
C07182=1168.450,-53.061,-43.678,179.384,5.854,149.226
C07183=1168.445,-52.812,-43.689,179.386,5.855,149.226
C07184=1168.439,-52.562,-43.700,179.388,5.855,149.225
C07185=1168.435,-52.312,-43.711,179.391,5.856,149.225
C07186=1168.430,-52.062,-43.723,179.393,5.855,149.224
C07187=1168.424,-51.813,-43.734,179.395,5.856,149.223
C07188=1168.419,-51.564,-43.745,179.397,5.857,149.223
C07189=1168.414,-51.313,-43.757,179.400,5.857,149.222
C07190=1168.408,-51.064,-43.768,179.402,5.857,149.222
C07191=1168.403,-50.814,-43.779,179.404,5.858,149.221
C07192=1168.398,-50.565,-43.791,179.407,5.858,149.221
C07193=1168.393,-50.294,-43.803,179.409,5.859,149.220
C07194=1168.387,-50.024,-43.816,179.412,5.859,149.219
C07195=1168.381,-49.753,-43.828,179.415,5.860,149.218
C07196=1168.376,-49.483,-43.841,179.417,5.860,149.218
C07197=1168.370,-49.233,-43.851,179.419,5.861,149.217
C07198=1168.365,-48.983,-43.863,179.422,5.860,149.217
C07199=1168.360,-48.733,-43.874,179.424,5.861,149.216
C07200=1168.355,-48.484,-43.886,179.426,5.862,149.215
C07201=1168.349,-48.235,-43.897,179.429,5.862,149.215
C07202=1168.344,-47.985,-43.909,179.431,5.863,149.214
C07203=1168.339,-47.735,-43.920,179.433,5.862,149.214
C07204=1168.334,-47.485,-43.932,179.435,5.863,149.213
C07205=1168.329,-47.235,-43.943,179.438,5.864,149.212
C07206=1168.323,-46.986,-43.955,179.440,5.865,149.212
C07207=1168.318,-46.737,-43.966,179.443,5.865,149.211
C07208=1168.313,-46.487,-43.978,179.445,5.865,149.211
C07209=1168.308,-46.237,-43.989,179.447,5.865,149.210
C07210=1168.303,-45.987,-44.001,179.450,5.866,149.209
C07211=1168.297,-45.738,-44.012,179.452,5.867,149.209
C07212=1168.292,-45.488,-44.024,179.455,5.867,149.208
C07213=1168.287,-45.238,-44.036,179.457,5.868,149.208
C07214=1168.282,-44.989,-44.047,179.459,5.867,149.207
C07215=1168.276,-44.739,-44.059,179.461,5.868,149.206
C07216=1168.272,-44.489,-44.070,179.464,5.869,149.206
C07217=1168.266,-44.240,-44.082,179.467,5.869,149.205
C07218=1168.261,-43.990,-44.093,179.469,5.870,149.205
C07219=1168.256,-43.740,-44.105,179.471,5.869,149.204
C07220=1168.250,-43.490,-44.117,179.473,5.870,149.203
C07221=1168.245,-43.241,-44.128,179.476,5.871,149.203
C07222=1168.240,-42.991,-44.140,179.478,5.872,149.202
C07223=1168.235,-42.741,-44.152,179.480,5.872,149.202
C07224=1168.229,-42.492,-44.163,179.483,5.872,149.201
C07225=1168.224,-42.242,-44.175,179.485,5.872,149.200
C07226=1168.219,-41.992,-44.186,179.487,5.873,149.200
C07227=1168.214,-41.743,-44.199,179.490,5.874,149.199
C07228=1168.209,-41.493,-44.211,179.492,5.874,149.198
C07229=1168.204,-41.244,-44.222,179.495,5.874,149.198
C07230=1168.199,-40.994,-44.234,179.497,5.875,149.197
C07231=1168.193,-40.744,-44.246,179.499,5.875,149.197
C07232=1168.188,-40.494,-44.257,179.501,5.876,149.196
C07233=1168.182,-40.245,-44.268,179.504,5.876,149.195
C07234=1168.177,-39.995,-44.281,179.506,5.877,149.195
C07235=1168.173,-39.746,-44.292,179.509,5.877,149.194
C07236=1168.167,-39.496,-44.304,179.512,5.878,149.194
C07237=1168.162,-39.246,-44.316,179.513,5.878,149.193
C07238=1168.156,-38.996,-44.328,179.516,5.878,149.192
C07239=1168.152,-38.746,-44.339,179.518,5.879,149.192
C07240=1168.146,-38.497,-44.352,179.521,5.879,149.191
C07241=1168.141,-38.247,-44.364,179.523,5.880,149.191
C07242=1168.136,-37.998,-44.375,179.525,5.881,149.190
C07243=1168.131,-37.748,-44.387,179.528,5.881,149.189
C07244=1168.126,-37.498,-44.400,179.530,5.881,149.189
C07245=1168.120,-37.248,-44.411,179.532,5.882,149.188
C07246=1168.115,-36.999,-44.422,179.535,5.882,149.187
C07247=1168.110,-36.749,-44.434,179.537,5.883,149.187
C07248=1168.105,-36.500,-44.447,179.540,5.883,149.186
C07249=1168.099,-36.250,-44.459,179.542,5.884,149.186
C07250=1168.094,-36.001,-44.470,179.545,5.884,149.185
C07251=1168.089,-35.751,-44.483,179.546,5.884,149.185
C07252=1168.084,-35.501,-44.494,179.549,5.885,149.184
C07253=1168.078,-35.251,-44.506,179.552,5.885,149.183
C07254=1168.073,-35.001,-44.518,179.554,5.886,149.183
C07255=1168.069,-34.752,-44.530,179.557,5.887,149.182
C07256=1168.063,-34.503,-44.542,179.559,5.887,149.182
C07257=1168.058,-34.253,-44.554,179.561,5.888,149.181
C07258=1168.053,-34.003,-44.567,179.564,5.888,149.180
C07259=1168.047,-33.753,-44.579,179.566,5.888,149.180
C07260=1168.043,-33.504,-44.591,179.568,5.889,149.179
C07261=1168.037,-33.254,-44.602,179.570,5.889,149.179
C07262=1168.032,-33.004,-44.614,179.573,5.890,149.178
C07263=1168.027,-32.755,-44.627,179.576,5.890,149.177
C07264=1168.021,-32.505,-44.639,179.578,5.891,149.177
C07265=1168.016,-32.256,-44.651,179.581,5.892,149.176
C07266=1168.011,-32.006,-44.663,179.583,5.892,149.176
C07267=1168.006,-31.756,-44.675,179.585,5.892,149.175
C07268=1168.001,-31.507,-44.687,179.588,5.892,149.174
C07269=1167.996,-31.257,-44.699,179.590,5.893,149.174
C07270=1167.990,-31.008,-44.712,179.592,5.894,149.173
C07271=1167.985,-30.758,-44.724,179.595,5.894,149.172
C07272=1167.980,-30.509,-44.736,179.597,5.895,149.172
C07273=1167.974,-30.259,-44.748,179.600,5.895,149.171
C07274=1167.970,-30.009,-44.761,179.602,5.896,149.171
C07275=1167.965,-29.759,-44.772,179.605,5.897,149.170
C07276=1167.960,-29.510,-44.785,179.606,5.897,149.169
C07277=1167.955,-29.260,-44.797,179.609,5.897,149.169
C07278=1167.950,-29.010,-44.809,179.612,5.897,149.168
C07279=1167.944,-28.760,-44.821,179.614,5.898,149.168
C07280=1167.939,-28.511,-44.834,179.616,5.899,149.167
C07281=1167.934,-28.261,-44.846,179.619,5.900,149.166
C07282=1167.928,-28.012,-44.858,179.621,5.900,149.166
C07283=1167.923,-27.762,-44.870,179.623,5.901,149.165
C07284=1167.918,-27.513,-44.883,179.626,5.901,149.165
C07285=1167.913,-27.263,-44.895,179.629,5.902,149.164
C07286=1167.907,-27.013,-44.907,179.630,5.902,149.163
C07287=1167.903,-26.763,-44.920,179.633,5.902,149.163
C07288=1167.897,-26.513,-44.932,179.635,5.903,149.162
C07289=1167.892,-26.264,-44.945,179.638,5.903,149.162
C07290=1167.887,-26.014,-44.957,179.641,5.904,149.161
C07291=1167.882,-25.765,-44.969,179.643,5.905,149.160
C07292=1167.876,-25.515,-44.981,179.645,5.905,149.160
C07293=1167.871,-25.266,-44.994,179.648,5.906,149.159
C07294=1167.866,-25.016,-45.006,179.650,5.906,149.158
C07295=1167.861,-24.766,-45.019,179.653,5.907,149.158
C07296=1167.856,-24.516,-45.031,179.655,5.908,149.157
C07297=1167.851,-24.247,-45.044,179.658,5.908,149.157
C07298=1167.845,-23.977,-45.057,179.660,5.908,149.156
C07299=1167.839,-23.707,-45.072,179.663,5.909,149.155
C07300=1167.834,-23.437,-45.084,179.665,5.910,149.155
C07301=1167.828,-23.188,-45.097,179.668,5.910,149.154
C07302=1167.824,-22.938,-45.110,179.671,5.911,149.153
C07303=1167.818,-22.688,-45.122,179.673,5.911,149.153
C07304=1167.813,-22.439,-45.134,179.675,5.912,149.152
C07305=1167.808,-22.189,-45.147,179.678,5.913,149.152
C07306=1167.803,-21.940,-45.160,179.680,5.913,149.151
C07307=1167.797,-21.690,-45.172,179.682,5.913,149.150
C07308=1167.792,-21.440,-45.185,179.685,5.913,149.150
C07309=1167.787,-21.190,-45.198,179.687,5.914,149.149
C07310=1167.782,-20.941,-45.210,179.689,5.915,149.149
C07311=1167.777,-20.691,-45.222,179.692,5.915,149.148
C07312=1167.772,-20.442,-45.235,179.695,5.916,149.147
C07313=1167.767,-20.192,-45.248,179.697,5.916,149.147
C07314=1167.762,-19.942,-45.260,179.700,5.917,149.146
C07315=1167.756,-19.693,-45.273,179.702,5.918,149.146
C07316=1167.751,-19.443,-45.285,179.704,5.918,149.145
C07317=1167.746,-19.194,-45.298,179.707,5.919,149.144
C07318=1167.741,-18.944,-45.311,179.709,5.919,149.144
